Omron CX-Programmer project NewProject (CX-Programmer 9.61)

# PLC NODE_4: CS1H-H CPU67
I/O table (CPU CS1H-CPU67H): rack 0 slot 0 CS1W-ETN21(ETN21Mode); rack 0 slot 1 CS1W-PRM21; rack 0 slot 2 CS1W-PRM21; rack 0 slot 3 CS1W-PRM21; rack 0 slot 4 CS1W-PRM21

## Global symbols (name address type ; comment)
AUTOPAADRAG_P8001 D20042 UINT
AUTOPAADRAG_P8002 D20142 UINT
AUTOPAADRAG_P8003 D20242 UINT
AUTOPAADRAG_V8014 D20092 UINT
AUTOPAADRAG_V8024 D20192 UINT
AUTOPAADRAG_V8034 D20292 UINT
1052.02 BOOL  ; V8223_2_AUTO
1151.00 BOOL  ; V0941_MANUELL
1151.12 BOOL  ; V0941_MAN.COM.BIT
1151.15 BOOL  ; V0941_LUKKET
1206.00 BOOL  ; C101_IND_VST80_K2
1206.01 BOOL  ; C102_IND_VST80_K2
1206.02 BOOL  ; C103_IND_VST80_K2
1206.03 BOOL  ; C104_IND_VST80_K2
1206.04 BOOL  ; C105
1206.05 BOOL  ; C106
1206.06 BOOL  ; C107
1206.07 BOOL  ; C108
1301.15 BOOL  ; C85_CONTAINER
1321.06 BOOL  ; VST80_K3_UPROG_7
1321.07 BOOL  ; VST80_K3_UPROG_8
1350.00 BOOL  ; VST 80_K2_AUTOVASK_VALGT
1350.01 BOOL  ; VST 80_K2_AUTOVASK_NR 1 STARTER
1350.02 BOOL  ; VST 80_K2_AUTOVASK_NR 2 STARTER
1350.03 BOOL  ; VST 80_K2_AUTOVASK_NR 3 STARTER
1350.04 BOOL  ; VST 80_K2_AUTOVASK_NR 4 STARTER
1350.05 BOOL  ; VST 80_K2_AUTOVASK_NR 5 STARTER
1350.10 BOOL  ; AUTOVASK STARTER
1350.11 BOOL  ; VST 80_K2_STARTIMPULS
1350.12 BOOL  ; AUTOVASK START RESETTES
1360.00 BOOL  ; AUTOVASK ER VALGT
1360.01 BOOL  ; VST 80_K3_AUTOVASK_NR 1 STARTER
1360.02 BOOL  ; VST 80_K3_AUTOVASK_NR 2 STARTER
1360.03 BOOL  ; VST 80_K3_AUTOVASK_NR 3 STARTER
1360.04 BOOL  ; VST 80_K3_AUTOVASK_NR 4  STARTER
1360.05 BOOL  ; VST 80_K3_AUTOVASK_NR 5 STARTER
1360.10 BOOL  ; VST 80_K3_AUTOVASK START. BIT SETTES FRA GRAFIKK
1360.11 BOOL  ; VST 80_K3_STARTIMPULS
1360.12 BOOL  ; Autovask Start Resettes
1402.13 BOOL  ; LL_T82_2_LUTTANK_2
1402.14 BOOL  ; HL_T82_2 Luttank 2
2100.05 BOOL  ; P2701.01 Toemming av T27.01
2100.06 BOOL  ; P2701.02 CIP Retur
2100.09 BOOL  ; P2701.01 Fylling av T27.01
2204.13 BOOL  ; V0416_UT
2204.15 BOOL  ; V0417_UT
2211.00 BOOL  ; V0416_OE_UT
2211.01 BOOL  ; V0416_N_UT
2211.02 BOOL  ; V0517_UT
2211.03 BOOL  ; V0701.19_UT
2211.08 BOOL  ; V8223_2_UT
2211.09 BOOL  ; V8224_2_UT
2212.00 BOOL  ; V0701.02_UT
2212.01 BOOL  ; V0701.03_UT
2212.02 BOOL  ; V0701.04_UT
2212.03 BOOL  ; V0701.05_UT
2212.04 BOOL  ; V0701.06_UT
2212.05 BOOL  ; V0701.07_UT
2212.06 BOOL  ; V0701.08_UT
2212.07 BOOL  ; V0701.10_UT
2212.08 BOOL  ; V0701.11_UT
2212.09 BOOL  ; V0701.12_UT
2212.10 BOOL  ; V0701.15_UT
2212.11 BOOL  ; V0701.24_UT
2212.12 BOOL  ; V0130_UT
2212.13 BOOL  ; V0131_UT
2212.14 BOOL  ; V0132_UT
2212.15 BOOL  ; V0133_UT
2213.00 BOOL  ; V0134_UT
2213.01 BOOL  ; V0135_UT
2213.02 BOOL  ; V0136_UT
2213.03 BOOL  ; V0137_UT
2213.04 BOOL  ; V0138_UT
2213.05 BOOL  ; V0231_UT
2213.06 BOOL  ; V0232_UT
2213.07 BOOL  ; V0233_UT
2213.08 BOOL  ; V0234_UT
2213.09 BOOL  ; V0235_UT
2213.10 BOOL  ; V0236_UT
2213.11 BOOL  ; V0237_UT
2213.12 BOOL  ; V0238_UT
2213.13 BOOL  ; V0701.13_UT
2213.14 BOOL  ; V0701.09_UT
2213.15 BOOL  ; V0701.14_UT
2214.14 BOOL  ; V0516_UT
2217.14 BOOL  ; V8120_Hjelp
2226.05 BOOL  ; V0645_UT
2226.07 BOOL  ; Isvannsventil L1
2226.08 BOOL  ; Isvannsventil L2
2240.14 BOOL  ; Vannv. gr.matpumpe
2242.00 BOOL  ; V2370_UT
2242.01 BOOL  ; V2371_UT
2242.02 BOOL  ; V2372_UT
2242.03 BOOL  ; V2373_UT
2242.04 BOOL  ; V2374_UT
2242.05 BOOL  ; V2375_UT
2242.06 BOOL  ; V2376_UT
2242.07 BOOL  ; V2409_UT
2243.00 BOOL  ; V0645_UT_N5
2244.00 BOOL  ; V0316_UT
2244.01 BOOL  ; V0316_OE_UT
2244.02 BOOL  ; V0316_N_UT
2244.03 BOOL  ; V0317_UT
2244.04 BOOL  ; V0318_UT
2244.05 BOOL  ; V0132_OE_UT
2244.06 BOOL  ; V0132_N_UT
2244.07 BOOL  ; V0136_OE_UT
2244.08 BOOL  ; V0136_N_UT
2244.09 BOOL  ; V0232_OE_UT
2244.10 BOOL  ; V0232_N_UT
2244.11 BOOL  ; V0236_OE_UT
2244.12 BOOL  ; V0236_N_UT
2244.13 BOOL  ; V0701.02_OE_UT
2244.14 BOOL  ; V0701.02_N_UT
2244.15 BOOL  ; V8016_UT
2245.00 BOOL  ; V0701.16_UT
2245.01 BOOL  ; V0701.17_UT
2245.02 BOOL  ; V0701.18_UT
2245.03 BOOL  ; V0702.01_UT
2245.04 BOOL  ; V0702.02_UT
2245.05 BOOL  ; V0702.03_UT
2245.06 BOOL  ; V0702.04_UT
2245.07 BOOL  ; V0702.06_UT
2245.08 BOOL  ; V0702.07_UT
2245.09 BOOL  ; V0702.08_UT
2245.10 BOOL  ; V0702.09_UT
2245.11 BOOL  ; V0427_UT
2245.12 BOOL  ; V0437_UT
2245.13 BOOL  ; V0527_UT
2245.14 BOOL  ; V0537_UT
2245.15 BOOL  ; V0702.10_UT
2246.00 BOOL  ; V2702.01_UT
2246.01 BOOL  ; V2702.02_UT
2246.02 BOOL  ; V4021_UT
2246.03 BOOL  ; V2702.04_UT
2246.04 BOOL  ; V2702.05_UT
2246.05 BOOL  ; V2702.06_UT
2246.06 BOOL  ; V2702.07_UT
2246.07 BOOL  ; V2702.08_UT
2246.08 BOOL  ; V2702.60_UT
2246.09 BOOL  ; V2702.61_UT
2246.10 BOOL  ; V4019_UT
2246.11 BOOL  ; V2702.04_UT
2246.12 BOOL  ; V2702.04_OE_UT
2246.13 BOOL  ; V2702.04_N_UT
2246.14 BOOL  ; V2702.09_UT
2246.15 BOOL  ; V4022_UT
2247.00 BOOL  ; V2703.01_UT
2247.01 BOOL  ; V2703.02_UT
2247.02 BOOL  ; V2703.03_UT
2247.03 BOOL  ; V2703.04_UT
2247.04 BOOL  ; V2703.05_UT
2247.05 BOOL  ; V2703.06_UT
2247.06 BOOL  ; V2703.07_UT
2247.07 BOOL  ; V2703.08_UT
2247.08 BOOL  ; V2703.09_UT
2247.09 BOOL  ; V2703.60_UT
2247.10 BOOL  ; V2703.61_UT
2247.11 BOOL  ; V2713_UT
2247.12 BOOL  ; V2703.10_UT
2247.13 BOOL  ; V2703.11
2247.14 BOOL  ; V2710_OE_UT
2247.15 BOOL  ; V2710_N_UT
2252.13 BOOL  ; V0702.12_UT
2252.14 BOOL  ; V0702.13_UT
2253.07 BOOL  ; KOMM_AVL_KULEV:
2253.15 BOOL  ; KOMM_AVL_SKRAASETEV.
2256.00 BOOL  ; V0702.11_UT
2256.01 BOOL  ; V0509_UT
2256.02 BOOL  ; V0702.12_UT
2256.03 BOOL  ; V0702.13_UT
2256.04 BOOL  ; V2606_UT
2256.05 BOOL  ; V2607_UT
2256.06 BOOL  ; V2608_UT
2256.07 BOOL  ; V2609_UT
2256.08 BOOL  ; V2605_UT
2256.09 BOOL  ; V2703.12_UT
2256.10 BOOL  ; V2606_UT
2256.11 BOOL  ; V2607_UT
2256.12 BOOL  ; V2608_UT
2256.13 BOOL  ; V2609_UT
2256.14 BOOL  ; V4401_UT
2256.15 BOOL  ; V4402_UT
2257.02 BOOL  ; V0509_INN
2258.00 BOOL  ; V2702.03_UT
2258.01 BOOL  ; V2702.03_OE_UT
2258.02 BOOL  ; V2702.03_N_UT
2258.03 BOOL  ; V2702.02_N
2258.04 BOOL  ; V2702.02_OE
2258.05 BOOL  ; V2703.02_N
2258.06 BOOL  ; V2703.02_OE
2258.07 BOOL  ; V2701.01_UT
2258.08 BOOL  ; V2701.02_UT
2258.09 BOOL  ; V2701.03_UT
2258.10 BOOL  ; V2701.04_UT
2258.11 BOOL  ; V2701.05_UT
2258.12 BOOL  ; V2701.06_UT
2258.13 BOOL  ; V2701.07_UT
2258.14 BOOL  ; V2701.08_UT
2258.15 BOOL  ; V2701.09_UT
2259.00 BOOL  ; V2701.10_UT
2259.01 BOOL  ; V2701.11_UT
2259.02 BOOL  ; V2701.12_UT
2259.03 BOOL  ; V2701.60_UT
2259.04 BOOL  ; V2701.61_UT
2259.05 BOOL  ; V2701.80_UT
2259.06 BOOL  ; V2701.81_UT
2259.07 BOOL  ; V2701.02_UT_OEvre loeft
2259.08 BOOL  ; V2701.02_UT_Nedre loeft
2259.09 BOOL  ; V4506_UT
2259.10 BOOL  ; V4507_UT
2259.11 BOOL  ; V4508_UT
2292.00 BOOL  ; PLS_6_V1004.70_UT
2292.01 BOOL  ; PLS_6_V1004.71_UT
2292.02 BOOL  ; PLS_6_V1004.72_UT
2292.03 BOOL  ; PLS_6_V1004.73_UT
2292.04 BOOL  ; PLS_6_V1004.74_UT
2292.05 BOOL  ; PLS_6_V1004.75_UT
2292.06 BOOL  ; PLS_6_V1004.76_UT
2403.05 BOOL  ; STOPPE LUFTBLAASING K1
2403.06 BOOL  ; STOPP LUFTBLAASING KURS 2
2403.07 BOOL  ; Stopp P8011 Kurs 1
2403.08 BOOL  ; Stopp P8011 Kurs 2
2403.09 BOOL  ; Stopp P8012 Kurs 1
2403.10 BOOL  ; Stopp P8012 Kurs 2
2403.11 BOOL  ; Stopp P8030 Kurs 1
2403.12 BOOL  ; Stopp P8030 Kurs 2
2403.13 BOOL  ; Stopp P8031 Kurs 1
2403.14 BOOL  ; Stopp P8031 Kurs 2
2403.15 BOOL  ; KURS 1 LINJE 2.1 og 2.2
2404.05 BOOL  ; P2703.01_UT
2404.06 BOOL  ; P2703.02_UT
2404.08 BOOL  ; RV T2702_UT
2404.09 BOOL  ; RV_T2703_UT
2405.00 BOOL  ; KURS 2 LINJE 2.1 og 2.2
2501.11 BOOL  ; T82_2_HL
2504.13 BOOL  ; V0416_INN
2504.15 BOOL  ; V0417_INN
2511.00 BOOL  ; V0416_OE_INN
2511.01 BOOL  ; V0416_N_INN
2511.02 BOOL  ; V0517_INN
2511.03 BOOL  ; V0701.19_INN
2512.00 BOOL  ; V0701.02_INN
2512.01 BOOL  ; V0701.03_INN
2512.02 BOOL  ; V0701.04_INN
2512.03 BOOL  ; V0701.05_INN
2512.04 BOOL  ; V0701.06_INN
2512.05 BOOL  ; V0701.07_INN
2512.06 BOOL  ; V0701.08_INN
2512.07 BOOL  ; V0701.10_INN
2512.08 BOOL  ; V0701.11_INN
2512.09 BOOL  ; V0701.12_INN
2512.10 BOOL  ; V0701.15_INN
2512.11 BOOL  ; V0701.24_INN
2512.12 BOOL  ; V0130_INN
2512.13 BOOL  ; V0131_INN
2512.14 BOOL  ; V0132_INN
2512.15 BOOL  ; V0133_INN
2513.00 BOOL  ; V0134_INN
2513.01 BOOL  ; V0135_INN
2513.02 BOOL  ; V0136_INN
2513.03 BOOL  ; V0137_INN
2513.04 BOOL  ; V0138_INN
2513.05 BOOL  ; V0231_INN
2513.06 BOOL  ; V0232_INN
2513.07 BOOL  ; V0233_INN
2513.08 BOOL  ; V0234_INN
2513.09 BOOL  ; V0235_INN
2513.10 BOOL  ; V0236_INN
2513.11 BOOL  ; V0237_INN
2513.12 BOOL  ; V0238_INN
2513.13 BOOL  ; V0701.13_INN
2513.14 BOOL  ; V0701.09_INN
2513.15 BOOL  ; V0701.14_INN
2514.14 BOOL  ; V0516_INN
2525.02 BOOL  ; V0429_INN
2525.03 BOOL  ; V0439_INN
2525.04 BOOL  ; V0529_INN
2525.05 BOOL  ; V0539_INN
2526.05 BOOL  ; V0645_INN
2526.07 BOOL  ; Isvannsventil L1
2526.08 BOOL  ; Isvannsventil L2
2542.00 BOOL  ; V2370_AKTIVERT
2542.01 BOOL  ; V2371_AKTIVERT
2542.02 BOOL  ; V2372_AKTIVERT_INN
2542.03 BOOL  ; V2373_AKTIVERT
2542.04 BOOL  ; B2374_NEDRE
2542.05 BOOL  ; V2375_AKTIVERT
2542.06 BOOL  ; V2376_AKTIVERT
2543.00 BOOL  ; N5_V0645_INN
2544.00 BOOL  ; V0316_INN
2544.01 BOOL  ; V0316_OE_INN
2544.02 BOOL  ; V0316_N_INN
2544.03 BOOL  ; V0317_INN
2544.04 BOOL  ; V0318_INN
2544.05 BOOL  ; V0132_OE_INN
2544.06 BOOL  ; V0132_N_INN
2544.07 BOOL  ; V0136_OE_INN
2544.08 BOOL  ; V0136_N_INN
2544.09 BOOL  ; V0232_OE_INN
2544.10 BOOL  ; V0232_N_INN
2544.11 BOOL  ; V0236_OE_INN
2544.12 BOOL  ; V0236_N_INN
2544.13 BOOL  ; V0701.02_OE_INN
2544.14 BOOL  ; V0701.02_N_INN
2544.15 BOOL  ; V8016_INN
2545.00 BOOL  ; V0701.16_INN
2545.01 BOOL  ; V0701.17_INN
2545.02 BOOL  ; V0701.18_INN
2545.03 BOOL  ; V0702.01_INN
2545.04 BOOL  ; V0702.02_INN
2545.05 BOOL  ; V0702.03_INN
2545.06 BOOL  ; V0702.04_INN
2545.07 BOOL  ; V0702.06_INN
2545.08 BOOL  ; V0702.07_INN
2545.09 BOOL  ; V0702.08_INN
2545.10 BOOL  ; V0702.09_INN
2545.11 BOOL  ; V0427_INN
2545.12 BOOL  ; V0437_INN
2545.13 BOOL  ; V0527_INN
2545.14 BOOL  ; V0537_INN
2545.15 BOOL  ; V0702.10_INN
2546.00 BOOL  ; V2702.01_INN
2546.01 BOOL  ; V2702.02_INN
2546.02 BOOL  ; V4021_INN
2546.03 BOOL  ; V2702.04_INN
2546.04 BOOL  ; V2702.05_INN
2546.05 BOOL  ; V2702.06_INN
2546.06 BOOL  ; V2702.07_INN
2546.07 BOOL  ; V2702.08_INN
2546.08 BOOL  ; V2702.60_INN
2546.09 BOOL  ; V2702.61_INN
2546.10 BOOL  ; V4019_INN
2546.11 BOOL  ; V2702.04_INN
2546.14 BOOL  ; V2702.09_INN
2546.15 BOOL  ; V4022_INN
2547.00 BOOL  ; V2703.01_INN
2547.01 BOOL  ; V2703.02_INN
2547.02 BOOL  ; V2703.03_INN
2547.03 BOOL  ; V2703.04_INN
2547.04 BOOL  ; V2703.05_INN
2547.05 BOOL  ; V2703.06_INN
2547.06 BOOL  ; V2703.07_INN
2547.07 BOOL  ; V2703.08_INN
2547.08 BOOL  ; V2703.09_INN
2547.09 BOOL  ; V2703.60_INN
2547.10 BOOL  ; V2703.61_INN
2547.11 BOOL  ; V2713_INN
2547.12 BOOL  ; V2703.10_INN
2547.13 BOOL  ; V2703.11_INN
2556.00 BOOL  ; V0702.11_INN
2556.01 BOOL  ; V0509_INN
2556.02 BOOL  ; V0702.12_INN
2556.03 BOOL  ; V0702.13_INN
2556.04 BOOL  ; V2606_INN
2556.05 BOOL  ; V2607_INN
2556.06 BOOL  ; V2608_INN
2556.07 BOOL  ; V2609_INN
2556.08 BOOL  ; V2605_INN
2556.09 BOOL  ; V2703.12_INN
2556.10 BOOL  ; V2606_INN
2556.11 BOOL  ; V2607_INN
2556.12 BOOL  ; V2608_INN
2556.13 BOOL  ; V2609_INN
2556.14 BOOL  ; V4401_INN
2556.15 BOOL  ; V4402_INN
2558.00 BOOL  ; V2702.03_INN
2558.07 BOOL  ; V2701.01_INN
2558.08 BOOL  ; V2701.02_INN
2558.09 BOOL  ; V2701.03_INN
2558.10 BOOL  ; V2701.04_INN
2558.11 BOOL  ; V2701.05_INN
2558.12 BOOL  ; V2701.06_INN
2558.13 BOOL  ; V2701.07_INN
2558.14 BOOL  ; V2701.08_INN
2558.15 BOOL  ; V2701.09_INN
2559.00 BOOL  ; V2701.10_INN
2559.01 BOOL  ; V2701.11_INN
2559.02 BOOL  ; V2701.12_INN
2559.03 BOOL  ; V2701.60_INN
2559.04 BOOL  ; V2701.61_INN
2559.05 BOOL  ; V2701.80_INN
2559.06 BOOL  ; V2701.81_INN
2559.09 BOOL  ; V4506_INN
2559.10 BOOL  ; V4507_INN
2559.11 BOOL  ; V4508_INN
2592.00 BOOL  ; PLS_6_V1004.70_AKTIVERT
2592.01 BOOL  ; PLS_6_V1004.71_AKTIVERT
2592.02 BOOL  ; PLS_6_V1004.72_AKTIVERT
2592.03 BOOL  ; PLS_6_V1004.73_AKTIVERT
2592.04 BOOL  ; PLS_6_V1004.74_AKTIVERT
2592.05 BOOL  ; PLS_6_V1004.75_AKTIVERT
2592.06 BOOL  ; PLS_6_V1004.76_AKTIVERT
2605.00 BOOL  ; B2370_HJEMME
2605.01 BOOL  ; V2370_HJEMME
2605.02 BOOL  ; V2371_HJEMME
2605.03 BOOL  ; V2372_HJEMME
2605.04 BOOL  ; V2373_HJEMME
2605.05 BOOL  ; B2374_OEVRE
2605.06 BOOL  ; V2375_HJEMME
2605.07 BOOL  ; V2376_HJEMME
2605.08 BOOL  ; START GRISEFOR MOT BIL
2605.09 BOOL  ; STOPP GRISEFOR MOT BIL
2605.10 BOOL  ; NOEDSTOPP GRISEFOR MOT BIL
2605.11 BOOL  ; STOPPSIGNAL FRA FLOWMAALER GRISEFOR MOT BIL
2605.12 BOOL  ; Lampe grisefor start_stopp
2605.13 BOOL  ; Startsignal til Q4401
2607.04 BOOL  ; FEIL MAGNETROERVERK T20.37
2607.05 BOOL  ; DRIFT MAGNETROERVERK T20.37
2607.06 BOOL  ; DRIFT MAGNETROERVERK T20.36
2607.11 BOOL  ; FEIL MAGNETROERVERK T20.36
2703.03 BOOL  ; H2370
2704.06 BOOL  ; P2703.01_INN
2704.07 BOOL  ; P2703.02_INN
2704.08 BOOL  ; RV_T2702_INN
2704.09 BOOL  ; RV_T2703_INN
2704.10 BOOL  ; Drift Grundfoss-pumper
2704.11 BOOL  ; Feil paa Grundfoss-pumper
2705.05 BOOL  ; PLS 4-P1940 INN
2712.05 BOOL  ; PLS_6_H1004.70_AKTIVERT
2713.05 BOOL  ; PLS_6_B1004.70_AKTIVERT
2713.06 BOOL  ; PLS_6_B1004.71_AKTIVERT
2800.04 BOOL  ; TIL PLS 5
2817.10 BOOL  ; PLS 5-P1940 INN
2817.11 BOOL  ; PLS 5-P1940 UT
2817.12 BOOL  ; PLS 4-P2040 INN
2817.13 BOOL  ; PLS 5-P2040 UT
2817.14 BOOL  ; PLS 5-P2039 INN
2817.15 BOOL  ; PLS 5-P2039 UT
2820.15 BOOL  ; V0939_UT_TIL_PLS5
2825.00 BOOL  ; N5_V0408_OEVRE
2846.06 BOOL  ; Slange Grisefor til PLS 5
2860.00 BOOL  ; Drift_Vibrator_21.10.02
2860.01 BOOL  ; Stopp_Vibrator_21.10.02
2860.02 BOOL  ; Drift_Knuser_21.02
2860.03 BOOL  ; Stopp_Knuser_21.02
2860.04 BOOL  ; Start_stopp_Vibrator_21.10.02
2860.05 BOOL  ; Start_stopp_Knuser_21.02
2860.06 BOOL  ; Start_stopp_Utmater_21.04
2861.00 BOOL  ; Drift Vifte 21.01.01
2861.01 BOOL  ; Stopp Vifte 21.01.01
2861.02 BOOL  ; Drift Vibrator 21.01.02
2861.03 BOOL  ; Stopp Vibrator 21.01.02
2861.04 BOOL  ; Drift Vifte 21.10.01
2861.05 BOOL  ; Stopp Vifte 21.10.01
2861.06 BOOL  ; Start_stopp_Vifte_21.01.01
2861.07 BOOL  ; Start_stopp_Vibrator_21.01.02
2861.08 BOOL  ; Start_stopp_Vifte_21.10.01
2901.15 BOOL  ; N5_V0408_OEVRE
2902.02 BOOL  ; FRA_NODE_5
2902.05 BOOL  ; N5-Lavt hovedlufttrykk
2903.15 BOOL  ; PLS 4-P1940 UT
2904.04 BOOL  ; 4-RV C49
2905.13 BOOL  ; Klapr_C56
2905.15 BOOL  ; Klapr_C92
2919.06 BOOL  ; 5-Bypass Mikronisator
2919.07 BOOL  ; 5-2919.07
2919.08 BOOL  ; 5-2919.08
2919.09 BOOL  ; 5-2919.09
2919.10 BOOL  ; 5-2919.10
2923.13 BOOL  ; N5_V2006_UT
2935.06 BOOL  ; V4302_UT_N5
2935.13 BOOL  ; V4302 Forsinkelse
2937.01 BOOL  ; 5-P2040_UT
2940.00 BOOL  ; N5_T20.36 Tapping
2940.01 BOOL  ; N5_T20.37 Tapping
2941 CHANNEL  ; N5_NIVAA_T2036
2944 CHANNEL  ; N5_NIVAA_T20.37
2946.00 BOOL  ; Retn.1 fra N5
2946.01 BOOL  ; Retn.2 fra N5
2946.02 BOOL  ; Isv.alarm fra N5
2955.07 BOOL  ; OPEN_DREN
2955.08 BOOL  ; OPEN_DYREFOR
2956.07 BOOL  ; OPEN_DREN_26
2956.08 BOOL  ; OPEN_DYREFOR_26
2959.00 BOOL  ; N5_V0408_OEVRE
302.13 BOOL  ; C106_VALG
302.14 BOOL  ; C107_VALG
4813.13 BOOL  ; TRYKKOMSLAG DP3 SPERRET
5117 CHANNEL  ; PT L1-1
5118 CHANNEL  ; PT L1-2
5119 CHANNEL  ; PT L2-1
5161.03 BOOL  ; .
5172 CHANNEL  ; TT T07.01
5173 CHANNEL  ; PT T07.01
5174 CHANNEL  ; TT T07.02
5175 CHANNEL  ; PT T07.02
5432.02 BOOL  ; Lampe drift grisefortoemming
5588 CHANNEL  ; TEMP_T82_2
5589 CHANNEL  ; Temp Kommunalt avloep
5590 CHANNEL  ; PH Kommunalt avloep
5591 CHANNEL  ; Flow Kommunalt avloep
5592 CHANNEL  ; BRIX Kommunalt avloep
5593 CHANNEL  ; PT T82_2
5594 CHANNEL  ; B8203_2
5595 CHANNEL  ; B8016
5596 CHANNEL  ; B8026
5597 CHANNEL  ; B8036
5601.02 BOOL  ; ¨
5667.03 BOOL  ; ¨
5730.00 BOOL  ; 360802
5761.02 BOOL  ; ,
5824.04 BOOL  ; '
587.00 BOOL  ; PGM587_DRIFT
587.01 BOOL  ; PGM587_0-STATUS
587.02 BOOL  ; PGM587_1-STATUS
587.03 BOOL  ; PGM587_2-STATUS
587.04 BOOL  ; PGM587_FEIL
587.05 BOOL  ; PGM587_FEILTID
587.06 BOOL  ; PGM587_INDKON
587.07 BOOL  ; PGM587_START
587.09 BOOL  ; PGM587_STOPP
587.10 BOOL  ; PGM587_STARTIMP.
587.11 BOOL  ; PGM587_ONIMPULS
587.14 BOOL  ; PGM587_OFFIMPULS
587.15 BOOL  ; PGM587_IND.INNE
588.00 BOOL  ; PGM 588 DRIFT
588.01 BOOL  ; 0-Status PGM 588
588.02 BOOL  ; PGM 588 1-Status
588.03 BOOL  ; PGM 588 2-Status
588.04 BOOL  ; PGM 588 FEIL
588.05 BOOL  ; PGM 588 Feiltid
588.06 BOOL  ; PGM 588_IndKon
588.07 BOOL  ; PGM 588 START
588.09 BOOL  ; PGM 588_STOPP
588.11 BOOL  ; PGM 588_Onimpuls
588.14 BOOL  ; PGM 588_Offimpuls
588.15 BOOL  ; PGM 588 Individkontroll
589.00 BOOL  ; PGM 589_DRIFT
589.01 BOOL  ; PGM 589 0-Status
589.02 BOOL  ; PGM 589 1-Status
589.03 BOOL  ; PGM 589_2-Status
589.04 BOOL  ; PGM 589_FEIL
589.05 BOOL  ; PGM589_FEILTID
589.06 BOOL  ; PGM 589_INDKON
589.07 BOOL  ; PGM 589_START
589.09 BOOL  ; PGM 589_STOPP
589.11 BOOL  ; PGM 589_ONIMPULS
589.14 BOOL  ; PGM 589_Offimpuls
589.15 BOOL  ; PGM 589_INDIVIDKONTROLL
590.00 BOOL  ; PGM 590 DRIFT
590.01 BOOL  ; 0-Status PGM 590
590.02 BOOL  ; 1-Status PGM 590
590.03 BOOL  ; PGM 590 2-Status
590.04 BOOL  ; PGM 590 FEIL
590.05 BOOL  ; PGM 590 Feiltid
590.06 BOOL  ; PGM 590 IndKon
590.07 BOOL  ; PGM 590 Start
590.09 BOOL  ; PGM 590_STOPP
590.11 BOOL  ; PGM 590 ONIMPULS
590.14 BOOL  ; PGM 590 Offimpuls
590.15 BOOL  ; PGM 590 Individkontroll
591.00 BOOL  ; PGM 591 DRIFT
591.01 BOOL  ; PGM 591 0-Status
591.02 BOOL  ; PGM 591 1-Status
591.03 BOOL  ; PGM 591_2-Status
591.04 BOOL  ; PGM 591 FEIL
591.05 BOOL  ; PGM 591 Feiltid
591.06 BOOL  ; PGM 591_IndKon
591.07 BOOL  ; PGM 591_START
591.09 BOOL  ; PGM 591_STOPP
591.11 BOOL  ; PGM 591_Onimpuls
591.14 BOOL  ; PGM 591_Offimpuls
591.15 BOOL  ; PGM 591_Individkontroll
592.00 BOOL  ; PGM 592_DRIFT
592.01 BOOL  ; PGM 592 0-Status
592.02 BOOL  ; PGM 592 1-Status
592.03 BOOL  ; PGM 592 2-Status
592.04 BOOL  ; PGM 592 FEIL
592.05 BOOL  ; PGM 592 Feiltid
592.06 BOOL  ; PGM 592_IndKon
592.07 BOOL  ; PGM 592 Start
592.09 BOOL  ; PGM 592_FEILTID
592.11 BOOL  ; PGM 592_Onimpuls
592.14 BOOL  ; PGM 592_Offimpuls
592.15 BOOL  ; PGM 592_Individkontroll
593.00 BOOL  ; PGM 593 DRIFT
593.01 BOOL  ; PGM 593 0-Status
593.02 BOOL  ; PGM 593_1-Status
593.03 BOOL  ; PGM 593_2-Status
593.05 BOOL  ; PGM 593_Feiltid
593.06 BOOL  ; PGM 593 IndKon
593.07 BOOL  ; PGM 593_START
593.09 BOOL  ; PGM 593_STOPP
593.11 BOOL  ; PGM 593 Onimpuls
593.14 BOOL  ; PGM 593_Offimpuls
593.15 BOOL  ; PGM 593 Individkontroll
600.02 BOOL  ; Drenering C33
608.04 BOOL  ; UHT-Anlegg mot Dypvannsutslipp
609.00 BOOL  ; RV2703Y
609.01 BOOL  ; RV2703I
609.02 BOOL  ; T2703_Vasket
609.03 BOOL  ; T2703_ManStartet
609.04 BOOL  ; T27.02_Sperr
609.05 BOOL  ; T27.03_Sperr
609.06 BOOL  ; P270301_ManStartet
609.07 BOOL  ; P270302_ManStartet
609.08 BOOL  ; P270201_ManStartet
609.09 BOOL  ; T2702_Vasket
609.10 BOOL  ; P070201_ManStartet
609.11 BOOL  ; P270201_I
609.12 BOOL  ; P270201_Y
609.13 BOOL  ; RV2702Y
609.14 BOOL  ; RV2702I
609.15 BOOL  ; Manuell Ansep CIP
610.00 BOOL  ; RV2702_ManStartet
610.01 BOOL  ; T0702_Vasket
610.02 BOOL  ; RV2703_ManStartet
610.03 BOOL  ; Start PGM 591.00
610.04 BOOL  ; Start PGM 589.00
610.05 BOOL  ; Start PGM 588.00
610.06 BOOL  ; Start PGM 590.00
610.07 BOOL  ; RV2703Y
610.09 BOOL  ; Dren til Silo 3
610.10 BOOL  ; Dren til Silo 4
610.11 BOOL  ; Dren til Silo 5
610.12 BOOL  ; Hj1_V0516
610.13 BOOL  ; Hj1_V0416
610.14 BOOL  ; Hj1_V0316
610.15 BOOL  ; Hj1_B0701.11
611.00 BOOL  ; Bil 1_Silo 3
611.01 BOOL  ; Bil 1_Silo 4
611.02 BOOL  ; Bil 1_Silo 5
611.03 BOOL  ; Henger 1_Silo 3
611.04 BOOL  ; Henger 1_Silo 4
611.05 BOOL  ; Henger 1_Silo 5
611.06 BOOL  ; Bil 2_Silo 3
611.07 BOOL  ; Bil 2_Silo 4
611.08 BOOL  ; Bil 2_Silo 5
611.09 BOOL  ; Henger 2_Silo 3
611.10 BOOL  ; Henger 2_Silo 4
611.11 BOOL  ; Henger 2_Silo 5
611.12 BOOL  ; Hj1_Dren til Silo 3
611.13 BOOL  ; Hj1_Drenering fra T0701 til Silo 4
611.14 BOOL  ; Hj1_Drenering fra T0701 til Silo 5
611.15 BOOL  ; Start PGM 592.00
612.03 BOOL  ; Vannsp_T27.02_Start
612.04 BOOL  ; Vannsp_T27.02_Drift
612.05 BOOL  ; Vannsp_T27.02_Feil
612.06 BOOL  ; Vannsp_T27.03_Start
612.07 BOOL  ; Vannsp_T27.03_Drift
612.08 BOOL  ; Vannsp_T27.03_Feil
612.09 BOOL  ; Vannsp_T27.40_Start
612.10 BOOL  ; Vannsp_T27.40_Drift
612.11 BOOL  ; Vannsp_T27.40_Feil
612.12 BOOL  ; Vannsp_T27.41_Start
612.13 BOOL  ; Vannsp_T27.41_Drift
612.14 BOOL  ; Vannsp_T27.41_Feil
612.15 BOOL  ; Manuell testbryter
613.00 BOOL  ; PGM 588 Hj1
613.01 BOOL  ; Start PGM 593.00
613.02 BOOL  ; PGM 592 Hj1
613.03 BOOL  ; Toerrkj. P4501
613.04 BOOL  ; Overtrykk, stopp griseforpumpe
613.05 BOOL  ; Hj1_Overtrykk gr_pumpe
613.06 BOOL  ; Makstid VST80 KURS 1
613.07 BOOL  ; Makstid for VST80 KURS 2
613.08 BOOL  ; Makstid utloept VST80 KURS 3
613.09 BOOL  ; Hj1_Autovask_80K3
613.10 BOOL  ; Hj2_Autovask_80K3
613.11 BOOL  ; Hj3_Autovask_80K3
613.12 BOOL  ; Hj4_Autovask_80_K3
613.13 BOOL  ; Hj5_Autovask_80K3
613.15 BOOL  ; PGM501_KOMMANDO_KOE
614.09 BOOL  ; Hj1_Autovask_80K2
614.10 BOOL  ; Hj2_Autovask_80K2
614.12 BOOL  ; Hj4_Autovask_80K2
614.13 BOOL  ; Hj5_Autovask_80K2
614.14 BOOL  ; Sperr innlesning til koeregister
614.15 BOOL  ; PGM 502 KOMMANDO_KOE
615.00 BOOL  ; Hj._0-Status_C101,C102
615.01 BOOL  ; Hj.1-Status_C101
615.02 BOOL  ; Hj.1-Status_C102
615.03 BOOL  ; PGM587_VALG
615.04 BOOL  ; Hj1_PGM587
615.05 BOOL  ; Hj2_PGM587
615.06 BOOL  ; Hj3_PGM587
615.07 BOOL  ; Hj4_PGM587
615.08 BOOL  ; Hj5_PGM587
615.09 BOOL  ; Hj6_PGM587
615.10 BOOL  ; Hj7_PGM587_Steg 1
615.11 BOOL  ; Hj8_PGM587_Steg 2
615.12 BOOL  ; Hj9_PGM587_Steg 3
615.13 BOOL  ; Hj10_PGM587_Steg 4
615.14 BOOL  ; Dren T27.01 til T20.33-35
615.15 BOOL  ; Slangefeil Trakt UHT
616.00 BOOL  ; PGM502_IND_C106_VALG
616.01 BOOL  ; PGM502_IND_C107_VALG
616.02 BOOL  ; PGM 589_VALG
616.03 BOOL  ; Hj1_PGM589
616.04 BOOL  ; Hj2_PGM589
616.05 BOOL  ; Hj3_PGM589
616.06 BOOL  ; Hj4_PGM589
616.07 BOOL  ; Hj5_PGM589
616.10 BOOL  ; PGM502_IND_C33_VALG
616.11 BOOL  ; C33_Drenert
616.12 BOOL  ; C33_Vasket
616.13 BOOL  ; C33_Hj1
616.14 BOOL  ; C33_Hj2
616.15 BOOL  ; Hj1_C14_V0582
617.00 BOOL  ; Hj.1_1-Status_C103
617.01 BOOL  ; Hj.2_1-Status_C104
617.02 BOOL  ; Hj.3_1-Status_C104
617.03 BOOL  ; Hj.4_1-Status_C104
617.04 BOOL  ; T07.01_Sperr
617.05 BOOL  ; T07.02_Sperr
617.06 BOOL  ; PGM 591_VALG
617.07 BOOL  ; Hj1_PGM 591
617.08 BOOL  ; Hj2_PGM 591
617.09 BOOL  ; Hj3_PGM 591
617.10 BOOL  ; Hj4_PGM 591
617.11 BOOL  ; Hj5_PGM 591
617.12 BOOL  ; PGM 592_VALG
617.13 BOOL  ; PGM 593_VALG
617.14 BOOL  ; PGM588_VALG
618.00 BOOL  ; Stopp fra FT Q2703
618.01 BOOL  ; Noedstopp fra Panel Deponi
618.02 BOOL  ; Stoppknapp Panel Deponi
618.03 BOOL  ; Startknapp Panel Deponi
618.04 BOOL  ; Lampe Drift Panel Deponi
618.05 BOOL  ; Startsignal til FT Q2703
618.06 BOOL  ; Hj.4_1-Status_C104
618.07 BOOL  ; Hj.5_1-Status C104
618.12 BOOL  ; Hj1_T0701_Sperr
618.13 BOOL  ; Hj2_T0701_Sperr
618.14 BOOL  ; Hj1_T0702_Sperr
618.15 BOOL  ; Hj2_T0702_Sperr
619.00 BOOL  ; Ny morgendrenering aktivert
619.01 BOOL  ; Dren L1.1 Til Silo 3
619.02 BOOL  ; Dren L1.1 Til Silo 4
619.03 BOOL  ; Dren L1.1 Til Silo 5
619.04 BOOL  ; Dren L1.2 Til Silo 3
619.05 BOOL  ; Dren L1.2 Til Silo 4
619.06 BOOL  ; Dren L1.2 Til Silo 5
619.07 BOOL  ; Dren L2.1 Til Silo 3
619.08 BOOL  ; Dren L2.1 Til Silo 4
619.09 BOOL  ; Dren L2.1 Til Silo 5
619.10 BOOL  ; Dren L2.2 Til Silo 3
619.11 BOOL  ; Dren L2.2 Til Silo 4
619.12 BOOL  ; Dren L2.2 Til Silo 5
619.13 BOOL  ; Kveldsdrenering Startet
619.14 BOOL  ; Nivaa i T0701 over SP
620.00 BOOL  ; Kveldsdrenering L1.1 Startet
620.01 BOOL  ; Kveldsdrenering L1.2 Startet
620.02 BOOL  ; Kveldsdrenering L2.1 Startet
620.03 BOOL  ; Kveldsdrenering L2.2 Startet
620.04 BOOL  ; Morgendrenering utfoert L1.1
620.05 BOOL  ; Morgendrenering utfoert L1.2
620.06 BOOL  ; Morgendrenering utfoert L2.1
620.07 BOOL  ; Morgendrenering utfoert L2.2
620.08 BOOL  ; Morgendrenering Turbiditet L1.1 over SP
620.09 BOOL  ; Morgendrenering Turbiditet L1.2 over SP
620.10 BOOL  ; Morgendrenering Turbiditet L2.1 over SP
620.11 BOOL  ; Morgendrenering Turbiditet L2.2 over SP
620.12 BOOL  ; Kveldsdrenering utfoert L1.1
620.13 BOOL  ; Kveldsdrenering utfoert L1.2
620.14 BOOL  ; Kveldsdrenering utfoert L2.1
620.15 BOOL  ; Kveldsdrenering utfoert L2.2
621.00 BOOL  ; Hj1_PGM 590
621.01 BOOL  ; Hj2_PGM 590
621.02 BOOL  ; Hj3_PGM 590
621.03 BOOL  ; Hj4_PGM 590
621.04 BOOL  ; Hj5_PGM 590
621.05 BOOL  ; Hj2_PGM592
621.06 BOOL  ; Hj3_PGM 592
621.07 BOOL  ; Hj4_PGM 592
621.08 BOOL  ; Hj5_PGM 592
621.09 BOOL  ; Hj6_PGM 592
621.10 BOOL  ; Hj1_PGM 593
621.11 BOOL  ; Hj2_PGM 593
621.12 BOOL  ; Hj3_PGM 593
621.13 BOOL  ; Hj4_PGM 593
621.14 BOOL  ; Hj4_PGM 593
622.00 BOOL  ; Hj1_PGM 588
622.01 BOOL  ; Hj3_PGM 588
622.02 BOOL  ; Hj4_PGM 588
622.03 BOOL  ; Hj5_PGM 588
622.04 BOOL  ; Hj1_L1.1_Kveldsdrenering
622.05 BOOL  ; Hj1_L1.2_Kveldsdrenering
622.06 BOOL  ; Hj1_L2.1_Kveldsdrenering
622.07 BOOL  ; Hj1_L2.2_Kveldsdrenering
622.08 BOOL  ; Hj1_Toem_T07.01
622.09 BOOL  ; Toem T07.02
622.10 BOOL  ; Test_3
622.11 BOOL  ; Flow OK VST80 K1
622.13 BOOL  ; UHT Trakt Prioritet
622.14 BOOL  ; 80K2_timingOK
622.15 BOOL  ; 80K3_timingOK
623.00 BOOL  ; Avloepstank 1 Mottak Overloep
623.01 BOOL  ; Avloepstank 1 Mottak HL
623.02 BOOL  ; Avloepstank 1 Mottak LL
623.03 BOOL  ; Avloepstank 1 Mottak Drift
623.04 BOOL  ; Avloepstank 1 Mottak Pumpe 1
623.05 BOOL  ; Avloepstank 1 Mottak Pumpe 2
623.06 BOOL  ; Avloepstank 1 Mottak Overloepsvarsel
623.07 BOOL  ; Avloepstank 2 Mottak Kjeller Overloep
623.08 BOOL  ; Avloepstank 2 Mottak Kjeller HL
623.09 BOOL  ; Avloepstank 2 Mottak Kjeller LL
623.10 BOOL  ; Avloepstank 2 Mottak Kjeller Drift
623.11 BOOL  ; Avloepstank 2 Mottak Kjeller Pumpe 3
623.12 BOOL  ; Avloepstank 2 Mottak Kjeller Overloepsvarsel
623.13 BOOL  ; Feil paa en frekvensomformer kommunalt avloep
623.14 BOOL  ; Reset makstemp dypvannsutslipp
623.15 BOOL  ; Reset doegntid
624.00 BOOL  ; Ny Kveldsdrenering aktivert
624.01 BOOL  ; Dren utfoert, toem T07.01
624.02 BOOL  ; T07.01 toemt, vanndren mot Silo
624.03 BOOL  ; Nye drenering C33 aktivert
624.04 BOOL  ; Kveldsdrenering Turbiditet L1.1 under SP
624.05 BOOL  ; Kveldsdrenering Turbiditet L1.2 under SP
624.06 BOOL  ; Kveldsdrenering Turbiditet L2.1 under SP
624.07 BOOL  ; Kveldsdrenering Turbiditet L2.2 under SP
624.08 BOOL  ; Morgendrenering L1.1 Startet
624.09 BOOL  ; Morgendrenering L1.2 Startet
624.10 BOOL  ; Morgendrenering L2.1 Startet
624.11 BOOL  ; Morgendrenering L2.2 Startet
624.12 BOOL  ; Hj1_Kveldsdrenering L1.1
624.13 BOOL  ; Hj1_Kveldsdrenering L1.2
624.14 BOOL  ; Hj1_Kveldsdrenering L2.1
624.15 BOOL  ; Hj1_Kveldsdrenering L2.2
625.01 BOOL  ; C106_Hj1
625.02 BOOL  ; Nye drenstart L1.1
625.03 BOOL  ; Nye drenstart L1.2
625.04 BOOL  ; Nye drenstart L2.1
625.05 BOOL  ; Nye drenstart L2.2
625.06 BOOL  ; Kveldsdren mot Silo 3
625.07 BOOL  ; Kveldsdren mot Silo 4
625.08 BOOL  ; Kveldsdren mot Silo 5
625.09 BOOL  ; Autodren Raamelkslinjer og Batteri
625.12 BOOL  ; Hurtigvask VST80_K2
625.13 BOOL  ; Hurtigvask VST80_K3
625.14 BOOL  ; Autovask_K3_Av_Paa
625.15 BOOL  ; Autovask K2_Av_Paa
626.00 BOOL  ; Makstid morgendrenering L1.1
626.01 BOOL  ; Makstid Moprgendrenering L1.2
626.02 BOOL  ; Makstid Morgendrenering L2.1
626.03 BOOL  ; Makstid Morgendrenering L2.2
626.04 BOOL  ; PGM501_IND_C102_VALG
626.05 BOOL  ; PGM501_IND_C101_VALG
626.06 BOOL  ; PGM501_IND_C06_VALG
626.07 BOOL  ; PGM501_IND_C103_VALG
626.08 BOOL  ; PGM501_IND_C104_VALG
626.09 BOOL  ; PGM501_IND_C105_VALG
626.10 BOOL  ; PGM501_IND_C108_VALG
626.11 BOOL  ; PGM501_IND_C53_VALG
626.12 BOOL  ; PGM501_IND_C54_VALG
626.13 BOOL  ; PGM501_IND_C77_VALG
626.14 BOOL  ; PGM501_IND_C78_VALG
626.15 BOOL  ; PGM501_IND_C79_VALG
627.00 BOOL  ; PGM502_IND_C12_VALG
627.01 BOOL  ; PGM502_IND_C13_VALG
627.02 BOOL  ; PGM502_IND_C14_VALG
627.03 BOOL  ; PGM502_IND_C30_VALG
627.04 BOOL  ; PGM502_IND_C09_VALG
627.05 BOOL  ; PGM502_IND_C10_VALG
627.06 BOOL  ; PGM502_IND_C15_VALG
628.00 BOOL  ; VST80_K1_Trinn 2 Turbiditet
628.01 BOOL  ; VST80_K2_Trinn 2 Turbiditet
628.02 BOOL  ; VST80_K3_Trinn 2_Turbiditet
628.03 BOOL  ; Nivaa i T07.02 OK
628.04 BOOL  ; T27.03 Vasket
628.05 BOOL  ; C104 Vasket
628.06 BOOL  ; Deponi-roer drenert
628.07 BOOL  ; T07.02 Vasket
628.08 BOOL  ; RV T07.01 Vasket
628.09 BOOL  ; T07.01 Vasket
628.10 BOOL  ; T27.02 Vasket
628.11 BOOL  ; PGM592_Hj1
628.12 BOOL  ; Isvann Hoey Temp Retning 1
628.13 BOOL  ; Isvann Hoey Temp Retning 2
628.14 BOOL  ; Hj5_V8221
628.15 BOOL  ; Hj6_V8221
629.00 BOOL  ; Autovask_K2_Hj1
629.01 BOOL  ; Autovask K3 Hj1
629.02 BOOL  ; C102 Vasket
629.03 BOOL  ; Autovask K2 Hj1
629.04 BOOL  ; V4202_Hj1
629.05 BOOL  ; Turbiditet i forskyll K1
629.06 BOOL  ; Turbiditet i forskyll K2
629.07 BOOL  ; Turbiditet i forskyll K3
629.08 BOOL  ; Hj.4_VST80K3
629.09 BOOL  ; Hj.5_VST80K3
630.00 BOOL  ; Dren batteri L1.1
630.01 BOOL  ; Dren batteri L1.2
630.02 BOOL  ; Dren batteri L2.1
630.03 BOOL  ; Dren batteri L2.2
630.04 BOOL  ; Start drenering av batteri
630.05 BOOL  ; Batteri L1.1 i drenering
630.06 BOOL  ; Batteri L1.2 i drenering
630.07 BOOL  ; Batteri L2.1 i drenering
630.08 BOOL  ; Batteri L2.2 i drenering
630.13 BOOL  ; T82_2_Hj1
630.14 BOOL  ; T82_2_Hj2
630.15 BOOL  ; T82_2_SPERRING
631.00 BOOL  ; Kveldsdrenering_Start_L2.1
631.01 BOOL  ; L2_1_Startknapp
631.02 BOOL  ; L2.1 Drenering Startet
631.03 BOOL  ; L2.1 Drenering Utfoert
631.04 BOOL  ; L2.1 Vann i Linje
631.05 BOOL  ; L2.1 Melk i Linje
631.06 BOOL  ; Kveldsdrenering_Start_L2.2
631.07 BOOL  ; L2.2 Startknapp
631.08 BOOL  ; L2.2 Drenering Startet
631.09 BOOL  ; L2.2 Drenering Utfoert
631.10 BOOL  ; L2.2 Vann i Linje
631.11 BOOL  ; L2.2 Melk i Linje
631.13 BOOL  ; Start Drenering C33
631.14 BOOL  ; Drenering C33 Startet
631.15 BOOL  ; Drenering C33 Utfoert
632.00 BOOL  ; Kveldsdrenering_Start_L1.1
632.01 BOOL  ; L1_1_Startknapp
632.02 BOOL  ; L1.1 Drenering Startet
632.03 BOOL  ; L1.1 Drenering Utfoert
632.04 BOOL  ; L1.1 Vann i Linje
632.05 BOOL  ; L1.1 Melk i Linje
632.06 BOOL  ; Kveldsdrenering_Start_L1.2
632.07 BOOL  ; L1_2_Startknapp
632.08 BOOL  ; L1_2_Startet
632.09 BOOL  ; L1.2 Drenering Utfoert
632.10 BOOL  ; L1.2 Vann i Linje
632.11 BOOL  ; L1.2 Melk i Linje
632.12 BOOL  ; Vann i Linje C33
632.13 BOOL  ; Melk i Linje C33
633.00 BOOL  ; L1.1_Dren_Hj1
633.01 BOOL  ; L1.1_Dren_Hj2
633.02 BOOL  ; L1.2_Dren_Hj1
633.03 BOOL  ; L1.2_Dren_Hj2
633.04 BOOL  ; L2.1_Dren_Hj1
633.05 BOOL  ; L2.1_Dren_Hj2
633.06 BOOL  ; L2.2 Dren_Hj1
633.07 BOOL  ; L2.2_Dren_Hj2
633.08 BOOL  ; Dren L1.1 under batteri
633.09 BOOL  ; Dren L1.2 under batteri
633.10 BOOL  ; Dren L2.1 under batteri
633.11 BOOL  ; Dren L2.2 under batteri
633.12 BOOL  ; Dren L1.1 batteri utfoert
633.13 BOOL  ; Dren L1.2 batteri utfoert
633.14 BOOL  ; Dren L2.1 batteri utfoert
633.15 BOOL  ; Dren L2.2 batteri utfoert
634.00 BOOL  ; C33_Dren_1-Status_Hj1
634.01 BOOL  ; C33_Dren_1-Status_Hj2
634.02 BOOL  ; C33_Dren_2-Status_Hj3
634.03 BOOL  ; C33_Dren_2-Status_Hj4
634.04 BOOL  ; Drenkontroll_L1.1
634.05 BOOL  ; Drenkontroll_L1.2
634.06 BOOL  ; Drenkontroll_L2.1
634.07 BOOL  ; Drenkontroll_L2.2
634.08 BOOL  ; Drenkontroll_C33
634.09 BOOL  ; C33 i drift
634.10 BOOL  ; V0701.20_UT
634.11 BOOL  ; V0701.20_INN
634.12 BOOL  ; Forsinkelse LL T07.01
634.13 BOOL  ; Manuell kjoering V2161 Damp Pasteur 21
634.14 BOOL  ; Floetepumpe P26.01_Inn
634.15 BOOL  ; Floetepumpe P26.01 UT
635.00 BOOL  ; C33_Dren_1-Status Hj4
635.01 BOOL  ; C33_Dren_1-Status Hj5
635.02 BOOL  ; C33_Dren_1-Status Hj6
635.03 BOOL  ; Dren_Batteri
635.04 BOOL  ; Dren_Linjer
635.05 BOOL  ; T0701_Drift_Drenering
635.06 BOOL  ; Turbiditet_Over_SP L1.1
635.07 BOOL  ; Turbiditet_Over_SP_L1.2
635.08 BOOL  ; Turbiditet_Over_SP_L2.1
635.09 BOOL  ; Turbiditet_Over_SP_L2.2
635.10 BOOL  ; Ok aa drenere batteriet
635.11 BOOL  ; Ok aa drenere Linjene
635.12 BOOL  ; Makstid drenering L1.1
635.13 BOOL  ; Makstid for drenering L1.2
635.14 BOOL  ; Makstid for drenering L2.1
635.15 BOOL  ; Makstid for drenering L2.2
636.00 BOOL  ; Rele' drift til P2040
636.01 BOOL  ; P2040 Drift
636.02 BOOL  ; P1940 Drift
636.03 BOOL  ; Griseforpumpe P1940 Start
636.04 BOOL  ; Griseforpumpe manuell hast.
636.05 BOOL  ; P2040 Manuell hast.
636.06 BOOL  ; Floetepumpe P2039 Manuell hast.
636.07 BOOL  ; P2039_UT
636.08 BOOL  ; Start slange grisefor
636.09 BOOL  ; Slangedrift Skummesal
636.10 BOOL  ; Start slange grisefor 1-status
636.11 BOOL  ; Start slange grisefor 2-status
636.12 BOOL  ; V9026_UT
636.13 BOOL  ; V9026_INN
638.00 BOOL  ; Toerrkjoerings-sperre for P0101 ved toemming av tankbil L1.1
638.01 BOOL  ; Toerrkjoerings-sperre for P0111 ved toemming av tankbil L1.2
638.02 BOOL  ; Toerrkjoerings-sperre for P0201 ved toemming av tankbil L2.1
638.03 BOOL  ; Toerrkjoerings-sperre for P0211 ved toemming av tankbil L2.2
639.09 BOOL  ; Hj1_RV_T27.02
639.12 BOOL  ; St_Kjoeling_T27.02
639.13 BOOL  ; St_Kjoeling_T27.03
639.14 BOOL  ; Ok aa starte kjoeling T27.02
639.15 BOOL  ; Ok aa starte kjoeling T27.03
641.02 BOOL  ; 1-Status L1.1
641.03 BOOL  ; 2 Status L1.1
641.04 BOOL  ; Fe_L1.1_Silo
641.05 BOOL  ; Feiltid_L1.1_Silo
641.07 BOOL  ; StL1.1_Silo
641.11 BOOL  ; Fe_Drenbatteri_L1.1
641.12 BOOL  ; DrenStBatteri_L1.1
641.13 BOOL  ; DrenBatteri_L1.1
641.14 BOOL  ; S1Batteri_L1.1
641.15 BOOL  ; S2Batteri_L1.1
642.02 BOOL  ; 1-Status L1.1
642.03 BOOL  ; 2-Status L1.2
642.04 BOOL  ; Fe_L1.2_Silo
642.05 BOOL  ; Feiltid_L1.2_Silo
642.07 BOOL  ; StL1.2_Silo
642.11 BOOL  ; Fe_Drenbatteri_L1.2
642.12 BOOL  ; DrenStBatteri_L1.2
642.13 BOOL  ; DrenBatteri_L1.2
642.14 BOOL  ; S1Batteri_L1.2
642.15 BOOL  ; S2Batteri_L1.2
643.02 BOOL  ; 1-Status L2.1
643.03 BOOL  ; 2-Status L2.1
643.04 BOOL  ; Fe_L2.1_Silo
643.05 BOOL  ; Feiltid_L2.1
643.07 BOOL  ; StL2.1_Silo
643.11 BOOL  ; Fe_Drenbatteri_L2.1
643.12 BOOL  ; DrenStBatteri_L2.1
643.13 BOOL  ; DrenBatteri_L2.1
643.14 BOOL  ; S1Batteri_L2.1
643.15 BOOL  ; S2Batteri_L2.1
644.02 BOOL  ; 1-Status L2.2
644.03 BOOL  ; 2-Status L2.2
644.04 BOOL  ; Fe_L2.2_Silo
644.05 BOOL  ; Feiltid_L2.2
644.07 BOOL  ; StL2.2_Silo
644.11 BOOL  ; Fe_Drenbatteri_L2.2
644.12 BOOL  ; DrenStBatteri_L2.2
644.13 BOOL  ; DrenBatteri_L2.2
644.14 BOOL  ; S1Batteri_L2.2
644.15 BOOL  ; S2Batteri_L2.2
645.00 BOOL  ; Turbiditet over setpunkt
645.01 BOOL  ; Start dren L1.2
645.02 BOOL  ; Start dren L2.1
645.03 BOOL  ; Start dren L2.2
645.08 BOOL  ; Hj1_0-Status Batteri L1.1
645.09 BOOL  ; Hj1_0-Status Batteri L1.2
645.10 BOOL  ; Hj1_0-Status Batteri L2.1
645.11 BOOL  ; Hj1_0-Status Batteri L2.2
645.12 BOOL  ; Start autodren L1.1
645.13 BOOL  ; Start autodren L1.2
645.14 BOOL  ; Start autodren L2.1
645.15 BOOL  ; Start autodren L2.2
646.00 BOOL  ; Hj1_0-Status L1.1
646.01 BOOL  ; Hj2_0-Status L1.1
646.02 BOOL  ; Hj3_0-Status L1.1
646.03 BOOL  ; Hj1_1-Status L1.1
646.04 BOOL  ; Hj2_1-Status L1.1
646.05 BOOL  ; Hj3_1-Status L1.1
646.06 BOOL  ; Hj4_1-Status L1.1
646.07 BOOL  ; Hj1_2-Status L1.1
646.08 BOOL  ; Hj1_0-Status L1.2
646.09 BOOL  ; Hj2_0-Status L1.2
646.10 BOOL  ; Hj3_0-Satus L1.2
646.11 BOOL  ; Hj1_1-Status L1.2
646.12 BOOL  ; Hj2_1-Status L1.2
646.13 BOOL  ; Hj3_1-Status L1.2
646.14 BOOL  ; Hj4_1-Status L1.2
646.15 BOOL  ; Hj1_2-Status L1.2
647.00 BOOL  ; Hj1_0-Status L2.1
647.01 BOOL  ; Hj2_0-Status L2.1
647.02 BOOL  ; Hj3_0-Status L2.1
647.03 BOOL  ; Hj1_1-Status L2.1
647.04 BOOL  ; Hj2_1-Status L2.1
647.05 BOOL  ; Hj3_1-Status L2.1
647.06 BOOL  ; Hj4_1-Status L2.1
647.07 BOOL  ; Hj1_2-Status L2.1
647.08 BOOL  ; Hj1_0-Status L2.2
647.09 BOOL  ; Hj2_0-Status L2.2
647.10 BOOL  ; Hj3_0-Status L2.2
647.11 BOOL  ; Hj1_1-Status L2.2
647.12 BOOL  ; Hj2_1-Status L2.2
647.13 BOOL  ; Hj3_1-Status L2.2
647.14 BOOL  ; Hj4_1-Status L2.2
647.15 BOOL  ; Hj1_2-Status L2.2
650.04 BOOL  ; Hj.Ind.Inne_2_80K2
650.05 BOOL  ; C101_VALG_VST80K2
650.06 BOOL  ; C102_VALG_VST80K2
650.07 BOOL  ; C103_VALG_VST80_K2
650.08 BOOL  ; C104_VALG_VST80_K2
650.09 BOOL  ; C105_VALG_VST80_K2
650.10 BOOL  ; C108_VALG_VST80_K2
650.15 BOOL  ; Lavt damptrykk
651.02 BOOL  ; 1 status
651.03 BOOL  ; 2 status
651.04 BOOL  ; feil
651.07 BOOL  ; Roed blink
659.00 BOOL  ; Dr_Autodren
659.01 BOOL  ; S0_Autodren
659.02 BOOL  ; S1_Autodren
659.03 BOOL  ; S2_Autodren
659.04 BOOL  ; Fe_Autodren
659.07 BOOL  ; St_Autodren
659.08 BOOL  ; Feiltid_Batteridrenering L1.1
659.09 BOOL  ; Feiltid_Batteridrenering_L1.2
659.10 BOOL  ; Feiltid_Batteridrenering_L2.1
659.11 BOOL  ; Feiltid_Batteridrenering_L2.2
659.12 BOOL  ; Hj1_T0701_Drift
659.14 BOOL  ; Hj2_Autodren
659.15 BOOL  ; Hj1_Autodren
660.00 BOOL  ; St_Overpumping_Til_T27.02
660.02 BOOL  ; S1_Overpumping_Til_T27.02
660.03 BOOL  ; S2_Overpumping_Til_T27.02
660.04 BOOL  ; Fe_Overpumping_Til_T27.02
660.05 BOOL  ; Dr_Overpumping_T27.02
660.06 BOOL  ; St_Overpumping_Til_T27.03
660.08 BOOL  ; S1_Overpumping_Til_T27.03
660.09 BOOL  ; S2_Overpumping_Til_T27.03
660.10 BOOL  ; Fe_Overpumping_Til_T27.03
660.11 BOOL  ; Dr_Overpumping_Til_T27.03
660.12 BOOL  ; Dren_Toem luftutskiller L1.1
660.13 BOOL  ; Dren_Toem luftutskiller L1.2
660.14 BOOL  ; Dren_Luftutskiller L2.1
660.15 BOOL  ; Dren_Luftutskiller L2.2
661.02 BOOL  ; S1_Kjoeling_T27.02
661.03 BOOL  ; S2_Kjoeling_T27.02
661.04 BOOL  ; Fe_Kjoeling_T27.02
661.05 BOOL  ; Dr_Kjoeling_T27.02
661.08 BOOL  ; S1_Kjoeling_T27.03
661.09 BOOL  ; S2_Kjoeling_T27.03
661.10 BOOL  ; Fe_Kjoeling_T27.03
661.11 BOOL  ; Dr_Kjoeling_T27.03
661.12 BOOL  ; T27.02 i koe
661.13 BOOL  ; T27.02 koe-start
661.14 BOOL  ; T27.03 i koe
661.15 BOOL  ; T27.03 i koe-start
662.00 BOOL  ; V2702.08_UT
662.01 BOOL  ; V2703.13_UT
662.02 BOOL  ; V2703.14_UT
662.03 BOOL  ; V2702.08_INN
662.04 BOOL  ; V2703.13_INN
662.05 BOOL  ; V2703.14_INN
662.06 BOOL  ; Turbiditet over min. VST80 Luttank
677.01 BOOL  ; AV_PAA_PIGGING
724.00 BOOL  ; T20.36 Tapping
724.01 BOOL  ; T20.37 Tapping
724.02 BOOL  ; Nivaa T20.36 mellom 40 og 50 000 liter
724.03 BOOL  ; Nivaa T20.36 mellom 30 og 40 000 liter
724.04 BOOL  ; Nivaa T20.36 mellom 25 og 30 000 liter
724.05 BOOL  ; Nivaa T20.36 mellom 20 og 25 000 liter
724.06 BOOL  ; Nivaa T20.36 mellom 6 og 20 000 liter
724.07 BOOL  ; Nivaa T20.37 mellom 40 og 50 000 liter
724.08 BOOL  ; Nivaa T20.37 mellom 30 og 40 000 liter
724.09 BOOL  ; Nivaa T20.37 mellom 25 og 30 000 liter
724.10 BOOL  ; Nivaa T20.37 mellom 20 og 25 000 liter
724.11 BOOL  ; Nivaa T20.37 mellom 6 og 20 000 liter
724.12 BOOL  ; Nivaa T20.36 under 6 000 liter stopp roerverk
724.13 BOOL  ; Nivaa T20.37 under 6 000 stopp roerverk
800.04 BOOL  ; Man Bactofors P2301
800.07 BOOL  ; C106 HJ1
800.08 BOOL  ; C107 HJ1
800.09 BOOL  ; C106 HJ 2
800.10 BOOL  ; C106 HJ3
800.12 BOOL  ; C107 HJ3
800.13 BOOL  ; C107 HJ4
800.14 BOOL  ; C106 HJ4
800.15 BOOL  ; C107 HJ5
801.00 BOOL  ; P0501_HJ5
801.07 BOOL  ; MANUELL KNAPP
802.00 BOOL  ; Manuell toemming silo
802.01 BOOL  ; Fra silo 3
802.02 BOOL  ; Fra silo 4
802.03 BOOL  ; Fra silo 5
802.04 BOOL  ; Til silo 3
802.05 BOOL  ; Til silo 4
802.06 BOOL  ; Til silo 5
803.00 BOOL  ; Ferdig sterilisert
803.01 BOOL  ; Ferdig sterilisert
803.02 BOOL  ; Ferdig sterilisert
803.03 BOOL  ; Trykkomslag_Pasteur 21
803.04 BOOL  ; Trykkomslag_Pasteur 22
803.05 BOOL  ; Trykkomslag_Pasteur 23
810.00 BOOL  ; Forsinkelse utloept Past.21 DP1
810.01 BOOL  ; Start forsinkelse Past.21 DP1
810.02 BOOL  ; Forsinkelse utloept Past.21 DP2
810.03 BOOL  ; Start forsinkelse Past.21 DP2
810.04 BOOL  ; Forsinkelse utloept Past.22 DP1
810.05 BOOL  ; Start forsinkelse Past.22 DP1
810.06 BOOL  ; Forsinkelse utloept Past.22 DP2
810.07 BOOL  ; Start forsinkelse Past.22 DP2
810.08 BOOL  ; Forsinkelse utloept Past.22 DP3
810.09 BOOL  ; Start forsinkelse Past. 22 DP3
810.10 BOOL  ; Reset tellere omslag pasteurer
820.00 BOOL  ; PLS_6_V1004.70_DEAKTIVERT
820.01 BOOL  ; PLS_6_V1004.71_DEAKTIVERT
820.02 BOOL  ; PLS_6_V1004.72_DEAKTIVERT
820.03 BOOL  ; PLS_6_V1004.73_DEAKTIVERT
820.04 BOOL  ; PLS_6_V1004.74_DEAKTIVERT
820.05 BOOL  ; PLS_6_V1004.75_DEAKTIVERT
820.06 BOOL  ; PLS_6_V1004.76_DEAKTIVERT
821.00 BOOL  ; P0701.01_UT
821.01 BOOL  ; V2371_DEAKTIVERT
821.02 BOOL  ; V2372_DEAKTIVERT
821.03 BOOL  ; V2373_DEAKTIVERT
821.04 BOOL  ; V2374_DEAKTIVERT
821.05 BOOL  ; V2375_DEAKTIVERT
821.06 BOOL  ; V2376_DEAKTIVERT
821.07 BOOL  ; B2370_INN
821.09 BOOL  ; V4302_UT_N5
821.10 BOOL  ; V4202 Forsinkelse
822.00 BOOL  ; Lampe omslag past.21
822.01 BOOL  ; Lampe omslag past.22
822.02 BOOL  ; Lampe omslag past.23
822.03 BOOL  ; Vannventil P2304
823.00 BOOL  ; Start P0701.01
823.01 BOOL  ; Drift P0701.01
823.02 BOOL  ; Oppheve sperring kurs 1
823.03 BOOL  ; Oppheve sperring kurs 2
823.05 BOOL  ; HL T07.01
823.06 BOOL  ; Start P0702.01
823.07 BOOL  ; LL T07.01
823.08 BOOL  ; HL T07.02
823.09 BOOL  ; LL T07.02
823.10 BOOL  ; Driftsignal fra P0702.01
823.11 BOOL  ; Motorvern P0702.01
904.03 BOOL  ; 0
905.09 BOOL  ; Man Bactofors
905.10 BOOL  ; Man Bactofors P2304
905.11 BOOL  ; Man Bactofors P2101
905.12 BOOL  ; Man Bactofors P2104
905.13 BOOL  ; Man Bactofors P2201
905.14 BOOL  ; Man Bactofors P2204
909.03 BOOL  ; Proeveuttak kommunalt avloep
925.10 BOOL  ; Toemming grisefortank til bil
925.15 BOOL  ; Telling ferdig fra flowmaaler Q4401
941.04 BOOL  ; HJ1_V8223_2_AUT
953.14 BOOL  ; ¨
955.13 BOOL  ; ¨
962.07 BOOL  ; Startknapp slange skummesal
962.08 BOOL  ; Start slange Grisefor Skummesal
962.09 BOOL  ; Drift Slange Grisefor Skummesal
964.11 BOOL  ; Manuell reset
964.12 BOOL  ; Manuell reset
964.13 BOOL  ; Test flowmaaler VST80 K3
965.00 BOOL  ; Man.sirk. Isv.tank
966.00 BOOL  ; FLOW KURS 1 OK
966.01 BOOL  ; FLOW K2 OK
966.02 BOOL  ; FLOW K3 OK
967.00 BOOL  ; VST80_K2_AUTOVASK
967.01 BOOL  ; Hjelpebit  VST80_K2_AUTOVASK
967.02 BOOL  ; Hjelpebit VST80_K2_AUTOVASK
967.05 BOOL  ; Hjelpebit VST 80_K3_AUTOVASK
967.06 BOOL  ; Hjelpebit VST 80_K3_AUTOVASK
967.07 BOOL  ; Hjelpebit VST 80_K3_AUTOVASK
969.00 BOOL  ; HJ_1_V8224_2
972.00 BOOL  ; OPEN_V4210
972.01 BOOL  ; OPEN_V4211
972.02 BOOL  ; OPEN_V4218
972.04 BOOL  ; OPEN_V4219
C0135 BOOL  ; Makstid for drenering C33 til T07.01
C0136 BOOL  ; Makstid Drenering C33
C0137 BOOL  ; Makstid Toem T07.01
C0138 BOOL  ; Makstid Vanndren mot Silo
C0139 BOOL  ; Holdetid foer Turbiditet er ute
C0231 BOOL  ; Drenstid L1.1
C0232 BOOL  ; Drenstid L1.2
C0233 BOOL  ; Drenstid L2.1
C0234 BOOL  ; Drenstid L2.2
C0235 BOOL  ; Forsink reset drenering av batteri
C0236 BOOL  ; Drenstid L1.1
C0237 BOOL  ; Drenstid Batteri L1.1
C0238 BOOL  ; Drenstid L1.2
C0239 BOOL  ; Drenstid Batteri L1.2
C0240 BOOL  ; Drenstid L2.1
C0241 BOOL  ; Drenstid Batteri L2.1
C0242 BOOL  ; Drenstid L2.2
C0243 BOOL  ; Drenstid Batteri L2.2
C0244 BOOL  ; Feiltid_Overpumping til T27.02
C0245 BOOL  ; Feiltid_Overpumping_Til_T27.03
C0246 BOOL  ; Feiltid_Kjoeling_T27.02
C0257 BOOL  ; Hindre toerrkjoering for P0101
C0258 BOOL  ; Hindre toerrkjoering for P0111
C0259 BOOL  ; Hindre toerrkjoering for P0201
C0260 BOOL  ; Hindre toerrkjoering for P0211
C0261 BOOL  ; RV T27.02 Intervall Stopp
C0262 BOOL  ; RV T27.02 Intervall Drift
C0263 BOOL  ; RV T27.03 Intervall Stopp
C0264 BOOL  ; RV T27.03 Intervall Drift
C0351 BOOL  ; Doegnreset for dypvannstemp
C0684 BOOL  ; Klapreteller C79
C0685 BOOL  ; Klapreteller
C0686 BOOL  ; PAUSETID KOMMUNAL SPYLING
C0687 BOOL  ; FORSINKELSE SKRAASETEVENTIL
C0688 BOOL  ; SPYLETID BRIXMAALER KOMMUNALT AVLOEP
C0690 BOOL  ; SEKUNDER AAPEN MOT DYPVANNSUTSLIPP TELLER NED FRA 3600
C0691 BOOL  ; TIMER AAPEN MOT DYPVANNSUTSLIPP TELLER NED FRA 3600
C0692 BOOL  ; SEKUNDER FYLLEVENTIL V0655 ER AAPEN PAA VANNSPARETANK
C0693 BOOL  ; TIMER FYLLEVENTIL V0655 ER AAPEN PAA VANNSPARETANK
C0715 BOOL  ; Makstid for vask utloept
C0716 BOOL  ; Makstid for vask utloept
C0717 BOOL  ; Makstid for vask utloept
C135 CHANNEL  ; Makstid til T07.01 sendes til Historian
C351 CHANNEL  ; Doegnteller dypvannsutslipp
D10148 CHANNEL  ; Skalering for bruk av Historian
D10154 CHANNEL  ; Skalering for bruk i Historian
D11101 CHANNEL  ; P
D11102 CHANNEL  ; I
D11103 CHANNEL  ; D
D15003 CHANNEL  ; Node 4.03
D15004 CHANNEL  ; Node 4.04
D15005 CHANNEL  ; Node 4.05
D15006 CHANNEL  ; Node 4.06
D15007 CHANNEL  ; Node 4.07
D15008 CHANNEL  ; Node 4.08
D15009 CHANNEL  ; Node 4.09
D15010 CHANNEL  ; Node 4.10
D15011 CHANNEL  ; Node 4.11
D15012 CHANNEL  ; Node 4.12
D15013 CHANNEL  ; Node 4.13
D15014 CHANNEL  ; Node 4.14
D15015 CHANNEL  ; Node 4.15
D15028 CHANNEL  ; Slavefeil Bus 4
D15029 CHANNEL  ; Diagnosefeil Bus 4
D15031 CHANNEL  ; Node 5.01
D15032 CHANNEL  ; Node 5.02
D15033 CHANNEL  ; Node 5.03
D15034 CHANNEL  ; Node 5.04
D15035 CHANNEL  ; Node 5.05
D15036 CHANNEL  ; Node 5.06
D15037 CHANNEL  ; Node 5.07
D15038 CHANNEL  ; Node 5.08
D15039 CHANNEL  ; Node 5.09
D15040 CHANNEL  ; Node 5.10
D15041 CHANNEL  ; Node 5.11
D15042 CHANNEL  ; Node 5.12
D15043 CHANNEL  ; Node 5.13
D15044 CHANNEL  ; Node 5.14
D15045 CHANNEL  ; Node 5.15
D15046 CHANNEL  ; Node 5.16
D15047 CHANNEL  ; Node 5.17
D15048 CHANNEL  ; Node 5.18
D15049 CHANNEL  ; Node 5.19
D15050 CHANNEL  ; Node 5.20
D15058 CHANNEL  ; Slavefeil Bus 5
D15059 CHANNEL  ; Diagnosefeil Bus 5
D15062 CHANNEL  ; Node 3.02
D15063 CHANNEL  ; Node 3.03
D15088 CHANNEL  ; Slavefeil Bus 3
D15089 CHANNEL  ; Diagnosefeil Bus 3
D15091 CHANNEL  ; Node 2.01
D15092 CHANNEL  ; Node 2.02
D15093 CHANNEL  ; Node 2.03
D15094 CHANNEL  ; Node 2.04
D15095 CHANNEL  ; Node 2.05
D15096 CHANNEL  ; Node 2.06
D15097 CHANNEL  ; Node 2.07
D15098 CHANNEL  ; Node 2.12
D15099 CHANNEL  ; Node 2.13
D15100 CHANNEL  ; Node 2.14
D15101 CHANNEL  ; Node 2.15
D15102 CHANNEL  ; Node 2.16
D15103 CHANNEL  ; Node 2.17
D15104 CHANNEL  ; Node 2.18
D15105 CHANNEL  ; Node 2.19
D15106 CHANNEL  ; Node 2.20
D15107 CHANNEL  ; Node 2.21
D15108 CHANNEL  ; Node 2.22
D15109 CHANNEL  ; Node 2.23
D15110 CHANNEL  ; Node 2.24
D15111 CHANNEL  ; Node 2.25
D15112 CHANNEL  ; Node 2.26
D15113 CHANNEL  ; Node 2.27
D15118 CHANNEL  ; Slavefeil Bus 2
D15119 CHANNEL  ; Diagnosefeil Bus 2
D1658 CHANNEL  ; Temp Kommunalt avloep
D1660 CHANNEL  ; PH Kommunalt avloep
D1662 CHANNEL  ; Flow Kommunalt avloep
D1664 CHANNEL  ; Brix Kommunalt avloep
D1750 CHANNEL  ; Turbiditet retur kurs 1
D17500 CHANNEL  ; Turbiditet retur kurs 1
D1752 CHANNEL  ; Turbiditet retur kurs 2
D17520 CHANNEL  ; Turbiditet retur kurs 2
D1754 CHANNEL  ; Turbiditet retur kurs 3
D1756 CHANNEL  ; Turbiditet retur kurs 3
D196 CHANNEL  ; D3174
D4032 CHANNEL  ; TEMP DYPVANNSUTSLIPP
D4034 CHANNEL  ; SKALERING
D4036 CHANNEL  ; SKALERT VERDI FOR TEMP DYPVANNSUTSLIPP
D4374 CHANNEL  ; Turbiditetsmaaler Raamelkslinje 2.2 Skalert
D4376 CHANNEL  ; Linje 2.2 Skalert verdi
D4380 CHANNEL  ; Turbiditetsmaaler Raamelkslinje 1.1
D4382 CHANNEL  ; Turbiditet Raamelkslinje 1.1
D4384 CHANNEL  ; Linje 1.1 Skalert verdi
D4386 CHANNEL  ; Turbiditetsmaaler Raamelkslinje 1.2
D4388 CHANNEL  ; Turbiditetsmaaler Raamelkslinje 1.2 Skalert
D4390 CHANNEL  ; Linje 1.2 Skalert verdi
D4392 CHANNEL  ; Turbiditetsmaaler Raamelkslinje 2.1
D4394 CHANNEL  ; Turbiditesmaaler Raamelkslinje 2.1 Skalert
D4396 CHANNEL  ; Linje 2.1 Skalert verdi
D4398 CHANNEL  ; Turbiditetsmaaler Raamelkslinje 2.2
D4400 CHANNEL  ; Turbiditetsmaaler Raamelkslinje 2.2 Skalert
D4402 CHANNEL  ; Linje 2.2 Skalert verdi
D4408 CHANNEL  ; Hastighet P0701.01
D4411 CHANNEL  ; B07.01.03
D4412 CHANNEL  ; B07.01.04
D4413 CHANNEL  ; B07.02.03
D4414 CHANNEL  ; B07.02.04
D4427 CHANNEL  ; NIVAA T07.02
D4434 CHANNEL  ; PT L1-1 B0107
D4440 CHANNEL  ; PT L1-2 B0117
D4446 CHANNEL  ; PT L2-1 B0207
D4452 CHANNEL  ; PT L2-2 B0217
D4458 CHANNEL  ; PT ISVANN L1 B0108
D4464 CHANNEL  ; PT ISVANN L2 B0208
D4466 CHANNEL  ; TRYKKDIFF L1.1
D4468 CHANNEL  ; TRYKKDIFF L1.2
D4470 CHANNEL  ; TRYKKDIFF L2.1
D4472 CHANNEL  ; TRYKKDIFF L2.2
D4474 CHANNEL  ; B07.01.04
D4500 CHANNEL  ; VST 80_K2_AUTOVASK FELLESREGISTER
D4501 CHANNEL  ; VST 80_K2_AUTOV_CNR_V1
D4502 CHANNEL  ; VST 80_K2_AUTOV_CNR_V2
D4503 CHANNEL  ; VST 80_K2_AUTOV_CNR_V3
D4504 CHANNEL  ; VST 80_K2_AUTOV_CNR_V4
D4505 CHANNEL  ; VST 80_K2_AUTOV_CNR_V5
D4600 CHANNEL  ; VST 80_K3_AUTOVASK FELLESREGISTER
D4601 CHANNEL  ; VST 80_K3_AUTOV_CNR_V1
D4602 CHANNEL  ; VST 80_K3_AUTOV_CNR_V2
D4603 CHANNEL  ; VST 80_K3_AUTOV_CNR_V3
D4604 CHANNEL  ; VST 80_K3_AUTOV_CNR_V4
D4605 CHANNEL  ; VST 80_K3_AUTOV_CNR_V5
D4700 CHANNEL  ; Temp Kommunalt avloep til Panel verksted
D4702 CHANNEL  ; pH Kommunalt avloep til Panel verksted
D4704 CHANNEL  ; Flow kommunalt avloep til Panel verksted
D4706 CHANNEL  ; Brix Kommunalt avloep til Panel Verksted
D4708 CHANNEL  ; Nivaa i Vannsparetank til Panel Verksted
D4710 CHANNEL  ; Flow Vannsparetank til Panel Verksted
D4712 CHANNEL  ; Makstemp dypvannsutslipp
D4714 CHANNEL  ; Mintemp dypvannsutslipp
D4716 CHANNEL  ; Resttid foer autoreset dypvannsutslipp
D5016 CHANNEL  ; PGM501_KOEPLASS_4
D5018 CHANNEL  ; PGM501_KOEPLASS_5
D5026 CHANNEL  ; PGM502_KOEPLASS_4
D5028 CHANNEL  ; PGM502_KOEPLASS_5
D5030 CHANNEL  ; Verdi C0302 til Historian
D5130 CHANNEL  ; 80K3_Vask_Dag
D5132 CHANNEL  ; 80K3_Vask_Mnd
D5134 CHANNEL  ; 80K3_Vask_Time
D5136 CHANNEL  ; 80K3_Vask_Min
D5138 CHANNEL  ; 80K2_Vask_Dag
D5140 CHANNEL  ; 80K2_Vask_Mnd
D5142 CHANNEL  ; 80K2_Vask_Time
D5144 CHANNEL  ; 80K2_Vask_Min
D5146 CHANNEL  ; Fellesregister for tidspunkt
D5300 CHANNEL  ; Bil 1
D5302 CHANNEL  ; Henger 1
D5304 CHANNEL  ; Bil 2
D5306 CHANNEL  ; Henger 2
D5432 CHANNEL  ; TT B0103
D5436 CHANNEL  ; TT B0104
D5502 CHANNEL  ; Status til Dreamreport
D5504 CHANNEL  ; Status til Dreamreport
D6052 CHANNEL  ; D6026
D6290 CHANNEL  ; Sperrekode for T07.01
D6291 CHANNEL  ; Kode aktivert T07.01
D6292 CHANNEL  ; Sperrekode for T07.02
D6293 CHANNEL  ; Kode aktivert T07.02
D6294 CHANNEL  ; Sperrekode for T27.02
D6295 CHANNEL  ; Kode aktivert T27.02
D6296 CHANNEL  ; Sperrekode for T27.03
D6297 CHANNEL  ; Kode aktivert T27.03
D6300 CHANNEL  ; Nivaa Avloepstank 1 Mottak
D6302 CHANNEL  ; Avloepstank 2 Mottak Kjeller Nivaa
D6304 CHANNEL  ; TT T27.02
D6308 CHANNEL  ; TT T27.02
D6310 CHANNEL  ; TT T27.03
D6312 CHANNEL  ; D6314
D6314 CHANNEL  ; TT T27.03
D6336 CHANNEL  ; P20.39 Hastighet
D6400 CHANNEL  ; Man Hast P2101 Bactofors
D6402 CHANNEL  ; Man Hast P2104 Bactofors
D6404 CHANNEL  ; Man Hast P2201 Bactofors
D6406 CHANNEL  ; Man Hast P2204 Bactofors
D6408 CHANNEL  ; Man Hast P2301 Bactofors
D6410 CHANNEL  ; Man Hast P2304 Bactofors
D6514 CHANNEL  ; B2106
D6530 CHANNEL  ; B2108
D6546 CHANNEL  ; P21_Diff_1
D6562 CHANNEL  ; P21_Diff_2
D6594 CHANNEL  ; B2330
D6614 CHANNEL  ; B2206
D6630 CHANNEL  ; B2208
D6646 CHANNEL  ; P22_Diff_1
D6662 CHANNEL  ; P22_Diff_2
D6678 CHANNEL  ; P22_Diff_3
D6694 CHANNEL  ; P22_Diff_ISv.
D6714 CHANNEL  ; B2306
D6730 CHANNEL  ; B2308
D6746 CHANNEL  ; P23_Diff_1
D6762 CHANNEL  ; P23_Diff_2
D6778 CHANNEL  ; P23_Diff_3
D6794 CHANNEL  ; P23_Diff_Isv.
D6800 CHANNEL  ; Hastighet P2040
D6806 CHANNEL  ; Hastighet P2040
D6808 CHANNEL  ; Hastighet P1940
D6900 CHANNEL  ; Hastighet P1940
D6902 CHANNEL  ; Skalert hastighet P1940
D7004 CHANNEL  ; Turbiditet VST80 Luttank
D7008 CHANNEL  ; Skalert verdi Turbiditet VST80 Luttank
D7716 CHANNEL  ; C101_TYPE_VASK
D7717 CHANNEL  ; C102_TYPE_VASK
D7718 CHANNEL  ; C103_TYPE_VASK
D7719 CHANNEL  ; C104_TYPE_VASK
D7736 CHANNEL  ; VASKESTATUS C101
D7737 CHANNEL  ; VASKESTATUS C102
D7738 CHANNEL  ; VASKESTATUS C103
D7739 CHANNEL  ; VASKESTATUS C104
D7741 CHANNEL  ; C105_TYPE_VASK
D7742 CHANNEL  ; C_TYPE_VASK
D7743 CHANNEL  ; C108_TYPE_VASK
D8080 CHANNEL  ; ID nummer fra Bil Kurs 1
D8082 CHANNEL  ; ID nummer fra Henger Kurs 1
D8084 CHANNEL  ; ID nummer fra Bil Kurs 2
D8086 CHANNEL  ; ID nummer fra Henger Kurs 2
D8090 CHANNEL  ; Bil Kurs 1
D8092 CHANNEL  ; Henger Kurs 1
D8094 CHANNEL  ; Bil 2
D8096 CHANNEL  ; Henger 2
D8250 CHANNEL  ; T82_2_SPERR_KODE_INN
D8251 CHANNEL  ; D82_2_SPERR_KODE_UT
D9012 CHANNEL  ; T82_2_ER_TEMP
D9016 CHANNEL  ; T82_2_NIVAA
D9018 CHANNEL  ; T82_2_NIVAA
D9430 CHANNEL  ; VASKESTATUS
D9432 CHANNEL  ; VASKESTATUS
T0158 BOOL  ; Feiltid Start Autodren
T0182 BOOL  ; Vent foer Turbiditet er ute
T0183 BOOL  ; Vent foer Turbiditet er ute
T0184 BOOL  ; Vent foer Turbiditet er ute
T0211 BOOL  ; Makstid for morgendrenering L1.1
T0212 BOOL  ; Makstid for morgendrenering L1.2
T0213 BOOL  ; Makstid for morgendrenering L2.1
T0214 BOOL  ; Makstid for morgendrenering L2.2
T0215 BOOL  ; Makstid for kveldsdrenering L1.1
T0216 BOOL  ; Makstid for kveldsdrenering L1.2
T0217 BOOL  ; Makstid for kveldsdrenering L2.1
T0218 BOOL  ; Makstid for kveldsdrenering L2.2
T0219 BOOL  ; Forsinkelse Turbiditet L1.1
T0220 BOOL  ; Forsinkelse Turbiditet L1.2
T0221 BOOL  ; Forsinkelse Turbiditet L2.1
T0222 BOOL  ; Forsinkelse Turbiditet L2.2
T0223 BOOL  ; Forsinkelse Turbiditet Kveldsdrenering L1.1
T0224 BOOL  ; Forsinkelse Turbiditet Kveldsdrenering L1.2
T0225 BOOL  ; Forsinkelse Turbiditet Kveldsdrenering L2.1
T0226 BOOL  ; Forsinkelse Turbiditet Kveldsdrenering L2.2
T0237 BOOL  ; V4202 Forsinkelse
T0242 BOOL  ; Hold foer stenging av V4205
T0243 BOOL  ; Hold foer stenging av V4202
T0252 BOOL  ; C33_Hj2_Forsink_Ut
T0253 BOOL  ; Makstid_Drenering_T07.01
T0254 BOOL  ; B2106
T0255 BOOL  ; B2108
T0256 BOOL  ; P21_Diff_1
T0257 BOOL  ; P21_Diff_2
T0258 BOOL  ; P21_Diff_Isv.
T0259 BOOL  ; B2206
T0260 BOOL  ; B2208
T0261 BOOL  ; P22_Diff_1
T0262 BOOL  ; P22_Diff_2
T0263 BOOL  ; P22_Diff_3
T0264 BOOL  ; P22_Diff_Isv.
T0265 BOOL  ; B2306
T0266 BOOL  ; B2308
T0267 BOOL  ; P23_Diff_1
T0268 BOOL  ; P23_Diff_2
T0269 BOOL  ; P23_Diff_3
T0270 BOOL  ; P23_Diff_Isv.
T0273 BOOL  ; Forsinkelse turbiditetskontroll
T0274 BOOL  ; Forsinkelse turbiditetskontroll
T0275 BOOL  ; Forsinkelse turbiditetskontroll
T0276 BOOL  ; Forsinkelse turbiditetskontroll
T0278 BOOL  ; Makstid drenering til T27.02/T27.03
T0279 BOOL  ; Makstid drenering L1.1
T0280 BOOL  ; Makstid drenering L1.2
T0281 BOOL  ; Makstid drenering L2.1
T0282 BOOL  ; Makstid drenering L2.2
T0283 BOOL  ; Dren L1.1 batteri makstid
T0284 BOOL  ; Dren L1.2 batteri makstid
T0285 BOOL  ; Dren L2.1 batteri makstid
T0286 BOOL  ; Dren L2.2 batteri makstid
T0287 BOOL  ; Forsinkelse LL T07.01
T0305 BOOL  ; Tid etter ventil stenger
T0306 BOOL  ; Tid etter ventil stenger
T0307 BOOL  ; Tid etter ventil stenger
T0308 BOOL  ; Tid etter ventil stenger
T0312 BOOL  ; Feiltid L1.1
T0313 BOOL  ; Feiltid Batteridrenering L1.1
T0314 BOOL  ; Feiltid L1.2
T0315 BOOL  ; Feiltid Batteridrenering L1.2
T0316 BOOL  ; Feiltid L2.1
T0317 BOOL  ; Feiltid Batteridrenering L2.1
T0318 BOOL  ; Feiltid L2.2
T0319 BOOL  ; Feiltid Batteridrenering L2.2
T0706 BOOL  ; Autovask forsinker startimpuls
T0731 BOOL  ; Maks tid aapen for V0701.10
T0732 BOOL  ; PGM587 FEILTID
T0734 BOOL  ; PGM 589 FEILTID
T0735 BOOL  ; PGM 593 FEILTID
T0736 BOOL  ; Fra T07.01 mot Silo 3, Drenstid
T0737 BOOL  ; Fra T07.01 mot Silo 4, Drenstid
T0738 BOOL  ; Fra T07.01 mot Silo 5, Drenstid
T0787 BOOL  ; PGM 588 Feiltid
T0847 BOOL  ; Drenering fra T0701 til Silo 3
T0848 BOOL  ; Drenering fra T0701 til Silo 4
T0849 BOOL  ; Drenering fra T0701 til Silo 5
T0850 BOOL  ; Spyletid paa V0701.07
T0975 BOOL  ; Dreneringstid Deponi
T0976 BOOL  ; TID OVERTRYKK GRISEFORPUMPE
T0977 BOOL  ; TID IKKE OVERTRYKK GRISEFORPUMPE
B0101_0_1000 D2004 REAL  ; 0=0GRADER   1000=100.0 GRADER
B0101_HJREG1 D6138 REAL
B0101_TT D1714 REAL  ; ZZ
B0102_0_1000 D2006 REAL  ; 0=0GRADER   1000=100.0 GRADER
B0102_HJREG1 D6140 REAL
B0102_TT D1694 REAL  ; Z
B0103_FC 2602.00 BOOL  ; Z
B0103_TT_ISVTUR D2044 WORD  ; TUR ISVANSTEMP TIL MOTTAK SKALERT
B0103_TT_ISVTUR_RAA D1724 WORD  ; TUR ISVANSTEMP TIL MOTTAK
B0104_TT_ISVRETUR D2046 WORD  ; RETUR ISVANSTEMP FRA MOTTAK SKALERT
B0104_TT_ISVRETUR_RAA D1726 WORD  ; RETUR ISVANSTEMP FRA MOTTAK
B0105_HL 2600.08 BOOL  ; Z
B0106_LL 2602.04 BOOL  ; Z
B0106_ML 2602.05 BOOL  ; Z
B0111_0_1000 D2104 REAL  ; 0=0GRADER   1000=100.0 GRADER
B0111_HJREG1 D6142 REAL
B0111_TT D1716 REAL  ; ZZ
B0112TT D1700 REAL  ; Z
B0112_0_1000 D2106 REAL  ; 0=0GRADER   1000=100.0 GRADER
B0112_HJREG1 D6144 REAL
B0113_FC 2602.01 BOOL  ; Z
B0115_HL 2600.09 BOOL  ; Z
B0116_LL 2602.06 BOOL  ; Z
B0116_ML 2602.07 BOOL  ; Z
B0201_0_1000 D2204 REAL  ; 0=0GRADER   1000=100.0 GRADER
B0201_HJREG1 D6146 REAL
B0201_TT D1718 REAL  ; ZZ
B0202_0_1000 D2206 REAL  ; 0=0GRADER   1000=100.0 GRADER
B0202_HJREG1 D6148 REAL
B0202_TT D1706 REAL  ; Z
B0203_FC 2602.02 BOOL  ; Z
B0205_HL 2600.10 BOOL  ; Z
B0206_LL 2602.08 BOOL  ; Z
B0206_ML 2602.09 BOOL  ; Z
B0211_0_1000 D2304 REAL  ; 0=0GRADER   1000=100.0 GRADER
B0211_HJREG1 D6150 REAL
B0211_TT D1720 REAL  ; ZZ
B0212_0_1000 D2306 REAL  ; 0=0GRADER   1000=100.0 GRADER
B0212_HJREG1 D6152 REAL
B0212_TT D1712 REAL  ; Z
B0213_FC 2602.03 BOOL  ; Z
B0215_HL 2600.11 BOOL  ; Z
B0216_LL 2602.10 BOOL  ; Z
B0216_ML 2602.11 BOOL  ; Z
B0301_LL 2600.13 BOOL  ; Z
B0302_TT_T03 D1730 WORD  ; INNGANGS0RD TEMP.
B0303_PT_T03 D1732 WORD  ; INNGANGSORD NIVAA
B0303_TT D6000 CHANNEL  ; Z
B0304_PT D6002 CHANNEL  ; Z
B0351_FC 2601.00 BOOL  ; Z
B0361_FC 2601.01 BOOL  ; Z
B0401_LL 2600.01 BOOL  ; Z
B0402_HL 2600.00 BOOL  ; Z
B0403_PT_T04 D1722 WORD  ; INNGANGSORD NIVAA
B0403_TT D6020 CHANNEL  ; Z
B0403_TT_INN D1748 REAL
B0404_PT D6022 CHANNEL  ; Z
B0404_PT_MAALT D6046 INT
B0501_LL 2600.03 BOOL  ; Z
B0502_TT_T05 D1740 WORD  ; INNGANGS0RD TEMP.
B0503_PT_T05 D1742 WORD  ; INNGANGSORD NIVAA
B0503_TT D6040 CHANNEL  ; Z
B0504_PT D6042 CHANNEL  ; Z
B0504_PT_MAALT D6026 INT
B0510_FC 2601.09 BOOL  ; Z
B0601_PT D6064 INT
B0603_PT_T06 D1746 CHANNEL
B0604_LL 2601.12 BOOL
B0605_FLOW D6074 INT  ; 0_1000
B0605_IMP 2603.00 BOOL  ; 10-LITERSIMPULS FRA FLOWMAALER B0605
B0605_LITER D6078 LINT  ; MENGE UT AV T06 I LITER
B0605_MAX_FLOW D6076 INT  ; 0_1000
B201504_PT D6015 CHANNEL  ; NIVAA T20.15    0-1000
B2101_FLT_1 D10100 REAL
B2101_FLT_2 D10102 REAL
B2101_PT D3100 WORD
B2102_FLT_1 D10104 REAL
B2102_FLT_2 D10106 REAL
B2102_PT D3102 WORD
B2103_FLT_1 D10108 REAL
B2103_FLT_2 D10110 REAL
B2103_PT D3104 WORD
B2104_FLT_1 D10112 REAL
B2104_FLT_2 D10114 REAL
B2104_PT D3106 WORD
B2105_NEDSKALERING NEDSKALERING
B2105_TT D3108 WORD
B2106_NEDSKALERING NEDSKALERING
B2106_TT D3110 WORD
B2107_NEDSKALERING NEDSKALERING
B2107_TT D3112 WORD
B2107_TT_HJ D3136 WORD  ; D3112 +/- 0,5 GRADER
B2108_FLOW 4502.15 BOOL
B2108_FLOW_ERVERDI D8112 UINT
B2108_FT D3114 WORD
B2108_FT_L_PR_T D4170 WORD  ; 0-20000
B2108_MENGDE_INN D1672 CHANNEL
B2108_NEDSKALER NEDSKALERING
B2110_HL 2600.14 BOOL  ; Z
B2110_LL 2600.15 BOOL
B2114_PT_FLT2 D10122 REAL
B2115_PT D3164 UINT  ; 0-7,00BAR
B2115_PT_FLT1 D10090 REAL
B2115_PT_FLT2 D10092 REAL
B2119_FL D6160 REAL  ; 0-1000,00
B2119_FLOW D6164 REAL  ; 0-20000 LITERPR TIME
B2119_FL_INN D6158 WORD  ; 0-1000
B2119_NEDSKALERING NEDSKALERING
B2120_FLOW D3590 INT  ; 0-1000
B2120_FLOW_NEDSKALER NEDSKALERING
B2120_FORV_OPNAADD 4802.12 BOOL
B2120_IMP 2603.14 BOOL  ; MAALER PLASSERT VED SJAKT
B2120_MENGDE D3624 DINT  ; MENGDE I LITER
B2120_RESET 4802.11 BOOL  ; RESET MENGDE UT PAA LINJE
B2121_0_7BAR D3156 REAL
B2121_0_7_BAR D3154 REAL
B2121_NEDSKALERING NEDSKALERING
B2121_PT D3160 WORD  ; TRYKK MELLOM P2103 OG SEP21
B2121_PT_FLT D3166 REAL  ; 0-1000
B2121_PT_FLT1 D10116 REAL
B2121_PT_FLT2 D10118 REAL
B2121_PT_mB D3176 INT
B2201_PT D3200 INT
B2201_PT_FLT1 D10030 REAL
B2201_PT_FLT2 D10032 REAL
B2202_PT D3202 INT
B2202_PT_FLT1 D10034 REAL
B2202_PT_FLT2 D10036 REAL
B2203_PT D3204 INT
B2203_PT_FLT1 D10038 REAL
B2203_PT_FLT2 D10040 REAL
B2204_PT D3206 INT
B2204_PT_FLT1 D10042 REAL
B2204_PT_FLT2 D10044 REAL
B2205_NEDSKALERING NEDSKALERING
B2205_TT D3208 WORD
B2205_TT_INVERTERT D23014 WORD  ; TIL BRUK I REG V2252
B2206_NEDSKALERING NEDSKALERING
B2206_TT D3210 WORD
B2207_NEDSKALERING NEDSKALERING
B2207_TT D3212 WORD
B2207_TT_HJ D3256 WORD  ; D3212 +/- 0,5 GRADER
B2208_FT D3214 WORD  ; 0-1000
B2208_FT_L_PR_T D4270 WORD  ; 0-20000
B2208_MENGDE_INN D1674 CHANNEL
B2209_NEDSKALERING NEDSKALERING
B2209_TT D3312 WORD
B2210_HL 2601.14 BOOL  ; Z
B2210_LL 2601.15 BOOL
B2212_PT D3770 DINT
B2212_PT_FLT1 D10046 REAL
B2212_PT_FLT2 D10048 REAL
B2213_PT D3772 DINT
B2213_PT_FLT1 D10050 REAL
B2213_PT_FLT2 D10052 REAL
B2214_PT D3180 INT
B2214_PT_FLT1 D10124 REAL
B2214_PT_FLT2 D10126 REAL
B2215_PT D3298 UINT
B2215_PT_FLT1 D10086 REAL
B2215_PT_FLT2 D10088 REAL
B2219_FL D6260 REAL  ; 0-1000,00
B2219_FLOW D6264 REAL  ; 0-20000 LITERPR TIME
B2219_FL_INN D6258 WORD  ; 0-1000
B2219_NEDSKALERING NEDSKALERING
B2220_FLOW D3592 INT  ; 0-1000
B2220_FLOW_NEDSKALERING NEDSKALERING
B2220_FORV_OPNAADD 4812.12 BOOL
B2220_IMP 2603.15 BOOL  ; MAALER PLASSERT VED SJAKT
B2220_MENGDE D3724 DINT  ; MENGDE I LITER
B2220_RESET 4812.11 BOOL  ; RESET MENGDE UT PAA LINJE
B2302_NEDSKALER NEDSKALERING
B2302_TT D3774 INT
B2305_NEDSKALERING NEDSKALERING
B2305_TT D3300 WORD
B2306_NEDSKALERING NEDSKALERING
B2306_TT D3302 WORD
B2307_NEDSKALERING NEDSKALERING
B2307_TT D3304 WORD
B2307_TT_HJ D3366 WORD  ; D3212 +/- 0,5 GRADER
B2308_FT D3306 WORD
B2308_FT_L_PR_T D4370 WORD  ; 0-8000
B2308_MENGDE_INN D1676 CHANNEL
B2310_NEDSKALER NEDSKALERING
B2310_PT D3308 WORD
B2311_HL_BLK 2603.06 BOOL
B2312_LL_BLK 2603.07 BOOL
B2320_PT D3776 DINT
B2320_PT_FLT1 D10054 REAL
B2320_PT_FLT2 D10056 REAL
B2321_PT D3778 DINT
B2321_PT_FLT1 D10058 REAL
B2321_PT_FLT2 D10060 REAL
B2322_PT D3780 DINT
B2322_PT_FLT1 D10062 REAL
B2322_PT_FLT2 D10064 REAL
B2323_PT D3782 DINT
B2323_PT_FLT1 D10066 REAL
B2323_PT_FLT2 D10068 REAL
B2324_PT D3784 DINT
B2324_PT_FLT1 D10070 REAL
B2324_PT_FLT2 D10072 REAL
B2325_PT D3786 DINT
B2325_PT_FLT1 D10074 REAL
B2325_PT_FLT2 D10076 REAL
B2326_PT D3788 DINT
B2326_PT_FLT1 D10078 REAL
B2326_PT_FLT2 D10080 REAL
B2327_PT D3790 DINT
B2327_PT_FLT1 D10082 REAL
B2327_PT_FLT2 D10084 REAL
B2330_Nedskaler NEDSKALERING
B2330_TT D3792 INT
B2331_BLK_LOKK 2603.05 BOOL
B2332_NEDSKALLERING NEDSKALERING
B2332_TT D3796 INT  ; TEMP VANNKRETS I PAST.REGULERINGSSLOEYFE
B2333_NEDAKALERING NEDSKALERING
B2333_TT D3794 INT
B2360_LL 2603.08 BOOL
B2401_LL 2603.04 BOOL
B2404_NEDSKALERING NEDSKALERING
B2404_PT D3310 WORD
B270102_LL 2603.10 BOOL
B2702_HL 2600.04 BOOL
B2702_LL 2600.05 BOOL
B2703_HL 2600.06 BOOL
B2703_LL 2600.07 BOOL
B4001_LL 2602.13 BOOL
B4002_HL 2602.12 BOOL
B4003_PT_T2740 D1860 CHANNEL  ; 0-1000
B4003_PT_T2740_RAA D1850 CHANNEL
B4004_TT_T2740 D1862 CHANNEL  ; 0-1000
B4004_TT_T2740_RAA D1852 CHANNEL
B4101_LL 2602.15 BOOL
B4102_HL 2602.14 BOOL
B4103_PT_T2741 D1864 CHANNEL  ; 0-1000
B4103_PT_T2741_RAA D1854 CHANNEL
B4104_TT_T2741 D1866 CHANNEL  ; 0-1000
B4104_TT_T2741_RAA D1856 CHANNEL
B4301_SLKONT_PR2 5117.06 BOOL  ; SLANGEKONTROLL TRAKT 42
B8011_CT D1606 REAL  ; Z COND. RET. KURS1 VST80
B8012_TT D1612 REAL  ; Z RETURTEMP VST80 KURS1
B8013_FC 2601.02 BOOL  ; Z
B8014_TT D1600 REAL  ; Z TEMP-TUR. KURS1 VST80
B8015_FC 2601.05 BOOL  ; Z
B8021_CT D1608 REAL  ; Z COND. RET. KURS2 VST80
B8022_TT D1614 REAL  ; Z RETURTEMP VST80 KURS2
B8023_FC 2601.03 BOOL  ; Z
B8024_TT D1602 REAL  ; Z TEMP-TUR. KURS2 VST80
B8025_FC 2601.06 BOOL  ; Z
B8031_CT D1610 REAL  ; Z COND. RET. KURS3 VST80
B8032_TT D1616 REAL  ; Z RETURTEMP VST80 KURS3
B8033_FC 2601.04 BOOL  ; Z
B8034_TT D1604 REAL  ; Z TEMP-TUR. KURS3 VST80
B8035_FC 2601.07 BOOL  ; Z
B8041_CT D1638 REAL  ; Z
B8045_FC 2601.08 BOOL  ; Z
B8101_PT D1634 REAL  ; Z
B8101_TEMP_T81 D1648 REAL
B8201_PT D1628 REAL  ; Z
B8202_TT D1630 REAL  ; Z
B8203_CT D1632 REAL  ; Z
B8301_PT D1622 REAL  ; Z
B8302_TT D1624 REAL  ; Z
B8303_CT D1626 REAL  ; Z
B8401_PT D1618 REAL  ; Z
B8402_TT D1620 REAL  ; Z
B8403_COND D1646 REAL
B8403_CT D1636 REAL  ; Z
B8403_INN 5563 INT
BANE1_GEIT 1451.04 BOOL  ; VED START AV VASK BANE1,VIL VANNVENTIL Vx30 SPERRES OG TIDEN I TR3 SPERRES    x=1-2-3
BANE2_GEIT 1452.04 BOOL  ; VED START AV VASK BANE2,VIL VANNVENTIL Vx30 SPERRES OG TIDEN I TR3 SPERRES      x=1-2-3
BANE3_GEIT 1453.04 BOOL  ; VED START AV VASK BANE3,VIL VANNVENTIL Vx30 SPERRES OG TIDEN I TR3 SPERRES      x=1-2-3
BIL01_0_STATUS 520.01 BOOL  ; XN4_BIL1_. Alle objekter som ikke betjenes er ok
BIL01_1_STATUS 520.02 BOOL  ; XN4_BIL1_. Alle utstyrte objekter i 1.fase er ok
BIL01_2_STAT 520.03 BOOL  ; X Alle utstyrte objekter er ok. Pgm = ok.
BIL01_DRIFT 520.00 BOOL  ; XN4_BIL1_ i drift
BIL01_FEIL 520.04 BOOL  ; XFeil
BIL01_FEILTID 520.05 BOOL  ; X
BIL01_HJ0 420.04 BOOL  ; X
BIL01_HJ1 420.05 BOOL  ; X
BIL01_INDIVID_INNE 520.15 BOOL  ; XIndividadresse er
BIL01_INDKON 520.06 BOOL  ; XKontr. at bare en individadresse er hoey.
BIL01_KOELES 320.14 BOOL  ; SPERR INNLESNING TIL KOE-REGISTER.
BIL01_KOEPLASS_1 D5200 CHANNEL  ; XFOERST I KOE
BIL01_KOEPLASS_2 D5202 CHANNEL  ; X
BIL01_KOEPLASS_3 D5204 CHANNEL  ; X
BIL01_KOMMANDO_KOE 320.15 BOOL  ; D3000 VERDI KAN OVERFOERES TIL KOE-REGISTER.
BIL01_OFF_IMP 520.14 BOOL  ; X
BIL01_ONIMPULS 520.11 BOOL  ; XN4_BIL1_Startimpuls for  program
BIL01_RESET 520.09 BOOL  ; XN4_BIL1. Stopp og nedkobling av programmet
BIL01_START 520.07 BOOL  ; Xprogram starter
BIL01_STARTIMPULS 520.10 BOOL  ; XN4_BIL1. Startimpuls.
BIL01_T03_IND 1220.00 BOOL  ; X
BIL01_T04_IND 1220.01 BOOL  ; XN4_BIL1_TIL_T04_INDIVID
BIL01_T05_IND 1220.02 BOOL  ; X
BIL01_TID_S T0520 BOOL  ; X
BIL01_TID_T 520 NUMBER
BIL01_TIL_T03_VALG 320.00 BOOL  ; INDIVIDVALG FRA KOEREGISTER.
BIL01_TIL_T04_VALG 320.01 BOOL  ; INDIVIDVALG FRA KOEREGISTER.
BIL01_TIL_T05_VALG 320.02 BOOL  ; INDIVIDVALG FRA KOEREGISTER.
BIL01_TMU_USIKRET 520.08 BOOL  ; TMU
BIL02_0_STATUS 522.01 BOOL  ; XN4_BIL1_. Alle objekter som ikke betjenes er ok
BIL02_1_STATUS 522.02 BOOL  ; XN4_BIL1_. Alle utstyrte objekter i 1.fase er ok
BIL02_2_STAT 522.03 BOOL  ; X Alle utstyrte objekter er ok. Pgm = ok.
BIL02_DRIFT 522.00 BOOL  ; XN4_BIL1_ i drift
BIL02_FEIL 522.04 BOOL  ; XFeil
BIL02_FEILTID 522.05 BOOL  ; X
BIL02_HJ0 422.04 BOOL  ; X
BIL02_HJ1 422.05 BOOL  ; X
BIL02_INDIVID_INNE 522.15 BOOL  ; XIndividadresse er
BIL02_INDKON 522.06 BOOL  ; XKontr. at bare en individadresse er hoey.
BIL02_KOEINLES D5228 CHANNEL  ; XINNLESNING AVKOMMANDOVERDIER FRA D3000
BIL02_KOELES 322.14 BOOL  ; SPERR INNLESNING TIL KOE-REGISTER.
BIL02_KOEPLASS_1 D5220 CHANNEL  ; XFOERST I KOE
BIL02_KOEPLASS_2 D5222 CHANNEL  ; X
BIL02_KOEPLASS_3 D5224 CHANNEL  ; X
BIL02_KOEPLASS_4 D5226 CHANNEL  ; X
BIL02_KOMMANDO_KOE 322.15 BOOL  ; D3000 VERDI KAN OVERFOERES TIL KOE-REGISTER.
BIL02_OFF_IMP 522.14 BOOL  ; X
BIL02_ONIMPULS 522.11 BOOL  ; XN4_BIL1_Startimpuls for  program
BIL02_RESET 522.09 BOOL  ; XN4_BIL1. Stopp og nedkobling av programmet
BIL02_START 522.07 BOOL  ; Xprogram starter
BIL02_STARTIMPULS 522.10 BOOL  ; XN4_BIL1. Startimpuls.
BIL02_T03_IND 1222.00 BOOL  ; X
BIL02_T04_IND 1222.01 BOOL  ; XN4_BIL1_TIL_T04_INDIVID
BIL02_T05_IND 1222.02 BOOL  ; X
BIL02_TID_S T0522 BOOL  ; X
BIL02_TID_T 522 NUMBER
BIL02_TIL_T03_VALG 322.00 BOOL  ; INDIVIDVALG FRA KOEREGISTER.
BIL02_TIL_T04_VALG 322.01 BOOL  ; INDIVIDVALG FRA KOEREGISTER.
BIL02_TIL_T05_VALG 322.02 BOOL  ; XINDIVIDVALG FRA KOEREGISTER.
BK_21_NIVAA D3158 CHANNEL
BK_22_NIVAA D3248 CHANNEL
BLAASETID_FOR T0009 BOOL
BLIK_TID1_S T0871 BOOL
BLIK_TID2_S T0872 BOOL
BLINK 999.01 BOOL  ; 0,5 SEKUNERS BINK
BLINK_HURTIG T0895 BOOL  ; 0.2S BLINK
BRYTER_HJ 960.15 BOOL
BUS_BLAAS_LAB 2824.02 BOOL
BUS_BLAAS_UHT 2824.03 BOOL
BUS_KNAPP_V4302 2935.05 BOOL
BUS_SIGN_VACUUM 2824.01 BOOL
Betinget_Omslag_DP3 202.01 BOOL
C01_IND_VST80_K1 1200.00 BOOL  ; Z
C01_STATUS D7620 CHANNEL  ; VASKESTATUS
C01_TYPE_VASK D7600 CHANNEL  ; VALG AV VASK SE EGEN TABELL
C01_VALG_VST80_K1 300.00 BOOL  ; Z
C02_IND_VST80_K1 1200.03 BOOL  ; Z
C02_STATUS D7623 CHANNEL  ; VASKESTATUS
C02_TYPE_VASK D7603 CHANNEL  ; VALG AV VASK SE EGEN TABELL
C02_VALG_VST80_K1 300.03 BOOL  ; Z
C03_06_C81_SYRE 1454.11 BOOL  ; VASKES BARE MED SYRE
C03_07_C81_FORL_FASE 1454.00 BOOL
C03_07_C81_HETVANN 1454.12 BOOL
C03_07_C81_LUT_SYRE 1454.10 BOOL
C03_07_C81_NOEDSTOPP 1454.02 BOOL
C03_07_C81_STOPP_TUR 1454.01 BOOL
C03_IND_VST80_K2 1201.00 BOOL  ; Z
C03_STATUS D7720 CHANNEL  ; VASKESTATUS
C03_TYPE_VASK D7700 CHANNEL  ; VALG AV VASK SE EGEN TABELL
C03_VALG_VST80_K2 301.00 BOOL  ; Z
C05_IND_VST80_K2 1201.03 BOOL  ; Z
C05_STATUS D7723 CHANNEL  ; VASKESTATUS
C05_TYPE_VASK D7703 CHANNEL  ; VALG AV VASK SE EGEN TABELL
C05_VALG_VST80_K2 301.03 BOOL  ; Z
C06_IND_VST80_K2 1201.06 BOOL  ; Z
C06_STATUS D7726 CHANNEL  ; VASKESTATUS
C06_TYPE_VASK D7706 CHANNEL  ; VALG AV VASK SE EGEN TABELL
C06_VALG_VST80_K2 301.06 BOOL  ; Z
C07_IND_VST80_K2 1201.07 BOOL  ; Z
C07_STATUS D7727 CHANNEL  ; VASKESTATUS
C07_TYPE_VASK D7707 CHANNEL  ; VALG AV VASK SE EGEN TABELL
C07_VALG_VST80_K2 301.07 BOOL
C08_IND_VST80_K2 1201.08 BOOL  ; Z
C08_STATUS D7728 CHANNEL  ; VASKESTATUS
C08_TYPE_VASK D7708 CHANNEL  ; VALG AV VASK SE EGEN TABELL
C08_VALG_VST80_K2 301.08 BOOL  ; Z
C09_0_ST_HJ1 933.07 BOOL
C09_0_ST_HJ2 933.08 BOOL
C09_0_ST_HJ3 933.09 BOOL
C09_0_ST_HJ4 933.10 BOOL
C09_10_0_ST_HJ1 933.15 BOOL
C09_10_15_2_HJ1 936.03 BOOL
C09_1_HJ1 935.01 BOOL
C09_1_HJ2 935.02 BOOL
C09_C10_1_HJ1 935.05 BOOL
C09_IND_VST80_K3 1202.04 BOOL  ; Z
C09_STATUS D7824 CHANNEL  ; VASKESTATUS
C09_TYPE_VASK D7804 CHANNEL  ; VALG AV VASK SE EGEN TABELL
C09_VALG 302.04 BOOL
C10_0_ST_HJ1 933.11 BOOL
C10_0_ST_HJ2 933.12 BOOL
C10_0_ST_HJ3 933.13 BOOL
C10_0_ST_HJ4 933.14 BOOL
C10_1_HJ1 935.03 BOOL
C10_1_HJ2 935.04 BOOL
C10_IND_VST80_K3 1202.05 BOOL  ; Z
C10_STATUS D7825 CHANNEL  ; VASKESTATUS
C10_TYPE_VASK D7805 CHANNEL  ; VALG AV VASK SE EGEN TABELL
C10_VALG 302.05 BOOL
C12_1_HJ1 935.06 BOOL
C12_1_HJ2 935.07 BOOL
C12_C33_36_1_HJ1 935.09 BOOL
C12_IND_VST80_K3 1202.00 BOOL  ; Z
C12_STATUS D7820 CHANNEL  ; VASKESTATUS
C12_TYPE_VASK D7800 CHANNEL  ; VALG AV VASK SE EGEN TABELL
C12_VALG 302.00 BOOL  ; Z
C13_1_HJ1 935.10 BOOL
C13_1_HJ2 935.11 BOOL
C13_34_37_1_HJ1 935.13 BOOL
C13_IND_VST80_K3 1202.01 BOOL  ; Z
C13_STATUS D7821 CHANNEL  ; VASKESTATUS
C13_TYPE_VASK D7801 CHANNEL  ; VALG AV VASK SE EGEN TABELL
C13_VALG 302.01 BOOL  ; Z
C14_1_HJ1 935.14 BOOL
C14_1_HJ2 935.15 BOOL
C14_C35_38_1_HJ1 936.01 BOOL
C14_IND_VST80_K3 1202.02 BOOL  ; Z
C14_STATUS D7822 CHANNEL  ; VASKESTATUS
C14_TYPE_VASK D7802 CHANNEL  ; VALG AV VASK SE EGEN TABELL
C14_VALG 302.02 BOOL  ; Z
C15_1_HJ1 936.04 BOOL
C15_1_HJ2 936.05 BOOL
C15_1_HJ3 940.01 BOOL
C15_HJ1 934.04 BOOL
C15_HJ2 934.09 BOOL
C15_HJ3 934.10 BOOL
C15_HJ4 934.15 BOOL
C15_IND_VST80_K3 1202.06 BOOL  ; Z
C15_STATUS D7826 CHANNEL  ; VASKESTATUS
C15_TYPE_VASK D7806 CHANNEL  ; VALG AV VASK SE EGEN TABELL
C15_VALG 302.06 BOOL  ; Z
C17_DRE_ETTER_C_N6 2842.01 BOOL
C18_DRE_ETTER_C_N6 2842.02 BOOL
C19_DRE_ETTER_C_N6 2842.03 BOOL
C20_DRE_ETTER_C_N6 2842.04 BOOL
C21_DREN_STARTET 760.00 BOOL
C21_DREN_UTFOERT 760.01 BOOL
C21_LITER_PRS_UT D3640 UDINT
C21_STARTET 760.02 BOOL
C21_UTFOERT 760.03 BOOL
C22_LITER_PRS_UT D3740 UDINT
C23_ACC_FORSK_TID D3321 WORD
C23_ACC_HETV_SIRK_TID D3341 WORD
C23_ACC_LUTSIRK_TID D3325 WORD
C23_ACC_LUTSKYLL_TID D3329 WORD
C23_ACC_SYRESIRK_TID D3333 WORD
C23_ACC_SYRESKYLL_TID D3337 WORD
C23_AV_BLK_FYLL 4504.14 BOOL  ; SIGNAL SOM SKAL BENYTTES  VED OPPFYLING AV BLK ETTER VASK.
C23_AV_BLK_FYLL_S T0887 BOOL  ; SIGNAL SOM SKAL BENYTTES  VED OPPFYLING AV BLK ETTER VASK.
C23_AV_BLK_FYLL_T 0887 NUMBER
C23_FORLENG_FASE 4504.07 BOOL  ; PAST21
C23_FORSKYLL 4503.01 BOOL  ; PAST21
C23_FORSKYLLTELLER_C C0086 BOOL
C23_FORSKYLLTELLER_S C86 CHANNEL
C23_FORST_TIL_VST80 4504.12 BOOL  ; PAST21  PAST22 OG 23 MAA VENTE
C23_HJ_LUTSKYLL_LUT_TID D3330 WORD
C23_HJ_REG_FORSK_TID D3322 WORD
C23_HJ_REG_HETV_SIRK_TID D3342 WORD
C23_HJ_REG_LUTSIRK_TID D3326 WORD
C23_HJ_REG_SYRESIRK_TID D3334 WORD
C23_HJ_REG_SYRESKYLL_TID D3338 WORD
C23_KLAP_ER_TRINNTELLER D3640 INT
C23_KLAP_ER_TRINNTELLER_N5 2845 INT
C23_KLAP_ER_TRINNTID D3636 INT
C23_KLAP_INNE_VST80_K4 4504.15 BOOL
C23_KLAP_PRS_TRINNTELLER D3638 INT
C23_KLAP_PRS_TRINNTID D3634 INT
C23_LUTSIRK_TID_S T0094 BOOL
C23_LUTSIRK_TID_T 0094 NUMBER
C23_LUT_INN 4503.09 BOOL  ; PAST21
C23_LUT_INN_KONS_1 4503.10 BOOL  ; PAST21
C23_LUT_SIRK 4503.11 BOOL  ; PAST21
C23_LUT_SKYLL 4503.14 BOOL  ; PAST21
C23_LUT_SYRE 4504.10 BOOL  ; PAST21
C23_LUT_UT 4503.12 BOOL  ; PAST21
C23_LUT_UT_KONS_0 4503.13 BOOL  ; PAST21
C23_PROD_TEKST D3622 INT  ; TIL GRAFIKK
C23_PRS_FORSK_MENGDE D3344 WORD
C23_PRS_FORSK_TID D3320 WORD  ; D3321
C23_PRS_HETV_SIRK_TID D3340 WORD
C23_PRS_LUTSIRK_TID D3324 WORD
C23_PRS_LUTSKYLL_TID D3328 WORD
C23_PRS_SYRESIRK_TID D3332 WORD
C23_PRS_SYRESKYLL_TID D3336 WORD
C23_RAP_COND_LUT D9158 CHANNEL  ; VASKERAPPORT CONDUKTIVITET I LUTFASEN
C23_RAP_COND_SYRE D9164 CHANNEL  ; VASKERAPPORT COND. I SYRESIRK. I SEKUNDER
C23_RAP_FLOW D9190 CHANNEL  ; VASKERAPPORT  FLOW I L/T
C23_RAP_HJ_COND_LUT D9159 CHANNEL  ; VASKERAPPORT CONDUKTIVITET I LUTFASEN HJ.FUNK.
C23_RAP_HJ_COND_SYRE D9165 CHANNEL  ; VASKERAPPORT CONDUKTIVITET I SYREFASEN HJ.FUNK.
C23_RAP_HJ_TEMP_HETV D9171 CHANNEL  ; VASKERAPPORT TEMP.HETVANNSIRK. HJ_FUNKSJON
C23_RAP_HJ_TEMP_LUT D9157 CHANNEL  ; VASKERAPPORT TEMP UT AV PASTEUR  I LUTFASEN HJ_FUNKSJON
C23_RAP_HJ_TEMP_SYRE D9163 CHANNEL  ; VASKERAPPORT TEMP UT AV PASTEUR ISYREFASEN HJ_FUNKSJON
C23_RAP_SEK_FS D9150 CHANNEL  ; VASKERAPPORT TID I FORSKYLLING I SEKUNDER
C23_RAP_SEK_LUT D9154 CHANNEL  ; VASKERAPPORT TID I LUTSIRK. I SEKUNDER
C23_RAP_SEK_SYRE D9160 CHANNEL  ; VASKERAPPORT TID I FORSKYLLING I SEKUNDER
C23_RAP_STATUS D9166 CHANNEL  ; ¨
C23_RAP_TEMP_HETV D9170 CHANNEL  ; VASKERAPPORT TEMP.HETVANNSIRK.
C23_RAP_TEMP_LUT D9156 CHANNEL  ; VASKERAPPORT TEMP UT AV PASTEUR  I LUTFASEN
C23_RAP_TEMP_SYRE D9162 CHANNEL  ; VASKERAPPORT TEMP UT AV PASTEUR ISYREFASEN
C23_RAP_TID_HETV D9168 CHANNEL  ; VASKERAPPORT TID HETVANNSIRK.
C23_STERILISER 4504.11 BOOL  ; PAST21
C23_STERIL_AVSLUTT 4504.01 BOOL  ; PAST21
C23_STERIL_OPPVARM 4503.15 BOOL
C23_STERIL_SIRK 4504.00 BOOL  ; PAST21
C23_STERIL_V2104_LAV_TEMP 4504.04 BOOL  ; PAST21
C23_STOPP_ETTER_VM 4504.09 BOOL  ; PAST21
C23_STOPP_I_FASE 4504.08 BOOL  ; PAST21 STANSER PUMPER OG TILFOERSEL BAV LUT-SYRE
C23_SYRE_INN 4503.03 BOOL  ; PAST21
C23_SYRE_INN_KONS_1 4503.04 BOOL  ; PAST21
C23_SYRE_MED_FORSKYLL 4504.06 BOOL  ; PAST21
C23_SYRE_SIRK 4503.05 BOOL  ; PAST21
C23_SYRE_SKYLL 4503.08 BOOL  ; PAST21
C23_SYRE_UT 4503.06 BOOL  ; PAST21
C23_SYRE_UT_KONS_0 4503.07 BOOL  ; PAST21
C23_TEKST_BILDE D4042 CHANNEL
C23_V2104_LAV_TEMP 4504.05 BOOL  ; PAST21
C23_VASKEPGM_DRIFT 4503.00 BOOL  ; PAST21 FORLOEP INNE
C23_VASKERAPP_OK 4505.03 BOOL
C23_VASKETRINN_TEKST D3620 INT
C23_VASK_ENDE 4504.13 BOOL  ; SIGNAL SOM SKAL BENYTTES  VED OPPFYLING AV BLK ETTER VASK
C23_VENT_INN_UT_VASKEM 4503.02 BOOL  ; 450303
C24_ACC_FORSK_TID D3421 WORD
C24_ACC_HETV_SIRK_TID D3441 WORD
C24_ACC_LUTSIRK_TID D3425 WORD
C24_ACC_LUTSKYLL_TID D3429 WORD
C24_ACC_SYRESIRK_TID D3433 WORD
C24_ACC_SYRESKYLL_TID D3437 WORD
C24_AV_BLK_FYLL 4514.14 BOOL  ; SIGNAL SOM SKAL BENYTTES  VED OPPFYLING AV BLK ETTER VASK.
C24_AV_BLK_FYLL_S T0888 BOOL  ; SIGNAL SOM SKAL BENYTTES  VED OPPFYLING AV BLK ETTER VASK.
C24_AV_BLK_FYLL_T 0888 NUMBER
C24_ER_FORSK_MENGDE D3446 WORD
C24_FORLENG_FASE 4514.07 BOOL  ; PAST22
C24_FORSKYLL 4513.01 BOOL  ; PAST22
C24_FORST_TIL_VST80 4514.12 BOOL  ; PAST22  PAST21 OG 23 MAA VENTE
C24_HC_HOY_FLOW 4814.04 BOOL
C24_HC_HOY_FLOW_AV 4814.05 BOOL  ; ¨
C24_HC_HOY_FLOW_REG_VERDI D3750 INT  ; AKTUELL RESTTID I AKTUELL FASE
C24_HJ_LUTSKYLL_LUT_TID D3430 WORD
C24_HJ_REG_FORSK_TID D3422 WORD
C24_HJ_REG_HETV_SIRK_TID D3442 WORD
C24_HJ_REG_LUTSIRK_TID D3426 WORD
C24_HJ_REG_SYRESIRK_TID D3434 WORD
C24_HJ_REG_SYRESKYLL_TID D3438 WORD
C24_KLAP_ER_TRINNTELLER D3760 INT
C24_KLAP_ER_TRINNTID D3756 INT
C24_KLAP_INNE_VST80_K4 4514.15 BOOL
C24_KLAP_PRS_TRINNTELLER D3758 INT
C24_KLAP_PRS_TRINNTID D3754 INT
C24_LUT_INN 4513.09 BOOL  ; ¨
C24_LUT_INN_KONS_1 4513.10 BOOL  ; PAST22
C24_LUT_SIRK 4513.11 BOOL  ; PAST22
C24_LUT_SKYLL 4513.14 BOOL  ; PAST22
C24_LUT_SYRE 4514.10 BOOL  ; PAST22
C24_LUT_UT 4513.12 BOOL  ; PAST22
C24_LUT_UT_KONS_0 4513.13 BOOL  ; PAST22
C24_PROD_TEKST D3722 INT  ; TIL  GRAFIKK
C24_PRS_FORSK_MENGDE D3444 WORD
C24_PRS_FORSK_TID D3420 WORD
C24_PRS_HETV_SIRK_TID D3440 WORD
C24_PRS_LUTSIRK_TID D3424 WORD
C24_PRS_LUTSKYLL_TID D3428 WORD
C24_PRS_SYRESIRK_TID D3432 WORD
C24_PRS_SYRESKYLL_TID D3436 WORD
C24_RAP_COND_LUT D9258 CHANNEL  ; VASKERAPPORT CONDUKTIVITET I LUTFASEN
C24_RAP_COND_SYRE D9264 CHANNEL  ; VASKERAPPORT COND. I SYRESIRK. I SEKUNDER
C24_RAP_FLOW D9290 CHANNEL  ; VASKERAPPORT  FLOW I L/T
C24_RAP_HJ_COND_LUT D9259 CHANNEL  ; VASKERAPPORT CONDUKTIVITET I LUTFASEN HJ.FUNK.
C24_RAP_HJ_COND_SYRE D9265 CHANNEL  ; VASKERAPPORT CONDUKTIVITET I SYREFASEN HJ.FUNK.
C24_RAP_HJ_TEMP_HETV D9271 CHANNEL  ; VASKERAPPORT TEMP.HETVANNSIRK. HJ_FUNKSJON
C24_RAP_HJ_TEMP_LUT D9257 CHANNEL  ; VASKERAPPORT TEMP UT AV PASTEUR  I LUTFASEN HJ_FUNKSJON
C24_RAP_HJ_TEMP_SYRE D9263 CHANNEL  ; VASKERAPPORT TEMP UT AV PASTEUR ISYREFASEN HJ_FUNKSJON
C24_RAP_SEK_FS D9250 CHANNEL  ; VASKERAPPORT TID I FORSKYLLING I SEKUNDER
C24_RAP_SEK_LUT D9254 CHANNEL  ; VASKERAPPORT TID I LUTSIRK. I SEKUNDER
C24_RAP_SEK_SYRE D9260 CHANNEL  ; VASKERAPPORT TID I FORSKYLLING I SEKUNDER
C24_RAP_STATUS D9266 CHANNEL  ; VASKERAPPORT STATUS          0=GODKJ.  1=DRIFTFORS.  2= IKKE GODKJ.
C24_RAP_TEMP_HETV D9270 CHANNEL  ; VASKERAPPORT TEMP.HETVANNSIRK.
C24_RAP_TEMP_LUT D9256 CHANNEL  ; VASKERAPPORT TEMP UT AV PASTEUR  I LUTFASEN
C24_RAP_TEMP_SYRE D9262 CHANNEL  ; VASKERAPPORT TEMP UT AV PASTEUR ISYREFASEN
C24_RAP_TID_HETV D9268 CHANNEL  ; VASKERAPPORT TID HETVANNSIRK.
C24_STERILISER 4514.11 BOOL  ; PAST22
C24_STERIL_AVSLUTT 4514.01 BOOL  ; PAST22
C24_STERIL_OPPVARM 4513.15 BOOL  ; PAST22
C24_STERIL_SIRK 4514.00 BOOL  ; PAST22
C24_STOPP_ETTER_VM 4514.09 BOOL  ; PAST22
C24_STOPP_I_FASE 4514.08 BOOL  ; PAST22   STANSER PUMPER OG TILFOERSEL BAV LUT-SYRE
C24_SYRE_INN 4513.03 BOOL  ; PAST22
C24_SYRE_INN_KONS_1 4513.04 BOOL  ; PAST22
C24_SYRE_MED_FORSKYLL 4514.06 BOOL  ; ¨
C24_SYRE_SIRK 4513.05 BOOL  ; PAST22
C24_SYRE_SKYLL 4513.08 BOOL  ; PAST22
C24_SYRE_UT 4513.06 BOOL  ; PAST22
C24_SYRE_UT_KONS_0 4513.07 BOOL  ; PAST22
C24_TEKST_BILDE D4192 CHANNEL
C24_TMU_HC_HOY_FLOW 4814.06 BOOL
C24_VASKEPGM_DRIFT 4513.00 BOOL  ; PAST22  FORLOEP INNE
C24_VASKERAPP_OK 4515.03 BOOL
C24_VASKETRINN_TEKST D3720 INT
C24_VASK_ENDE 4514.13 BOOL  ; SIGNAL SOM SKAL BENYTTES  VED OPPFYLING AV BLK ETTER VASK
C24_VENT_INN_UT_VASKEM 4513.02 BOOL  ; PAST22   PAST2 ELLER PAST23 FYLLES-TOEMMES FOR VASKEMIDDEL
C254_KLAP_INNE_VST80_K4 4514.15 BOOL
C25_ACC_FORSK_TID D3521 WORD
C25_ACC_HETV_SIRK_TID D3541 WORD
C25_ACC_LUTSIRK_TID D3525 WORD
C25_ACC_LUTSKYLL_TID D3529 WORD
C25_ACC_SYRESIRK_TID D3533 WORD
C25_ACC_SYRESKYLL_TID D3537 WORD
C25_AVSLUTTET 4824.01 BOOL
C25_AV_BLK_FYLL 4524.14 BOOL  ; SIGNAL SOM SKAL BENYTTES  VED OPPFYLING AV BLK ETTER VASK.
C25_AV_BLK_FYLL_S T0889 BOOL  ; SIGNAL SOM SKAL BENYTTES  VED OPPFYLING AV BLK ETTER VASK.
C25_AV_BLK_FYLL_T 0889 NUMBER
C25_BLK_NIV 4824.00 BOOL  ; V2309 STENGES
C25_ER_FORSK_MENGDE D3546 WORD
C25_FORLENG_FASE 4524.07 BOOL  ; PAST23
C25_FORSKYLL 4523.01 BOOL  ; PAST23
C25_FORST_TIL_VST80 4524.12 BOOL  ; PAST23  PAST21 OG 22 MAA VENTE
C25_HJ_LUTSKYLL_LUT_TID D3530 WORD
C25_HJ_REG_FORSK_TID D3522 WORD
C25_HJ_REG_HETV_SIRK_TID D3542 WORD
C25_HJ_REG_LUTSIRK_TID D3526 WORD
C25_HJ_REG_SYRESIRK_TID D3534 WORD
C25_HJ_REG_SYRESKYLL_TID D3538 WORD
C25_IND_VST80_K4 1205.00 BOOL  ; VASK PAST23
C25_KLAP_ER_TRINNTELLER D3860 INT
C25_KLAP_ER_TRINNTID D3856 INT
C25_KLAP_INNE_VST80_K4 4524.15 BOOL
C25_KLAP_PRS_TRINNTELLER D3858 INT
C25_KLAP_PRS_TRINNTID D3854 INT
C25_LUT_INN 4523.09 BOOL  ; PAST23
C25_LUT_INN_KONS_1 4523.10 BOOL  ; PAST23
C25_LUT_SIRK 4523.11 BOOL  ; PAST23
C25_LUT_SKYLL 4523.14 BOOL  ; PAST23
C25_LUT_SYRE 4524.10 BOOL  ; PAST23
C25_LUT_UT 4523.12 BOOL  ; PAST23
C25_LUT_UT_KONS_0 4523.13 BOOL  ; ¨
C25_PROD_TEKST D3822 INT  ; TIL  GRAFIKK
C25_PRS_FORSK_MENGDE D3544 WORD
C25_PRS_FORSK_TID D3520 WORD
C25_PRS_HETV_SIRK_TID D3540 WORD
C25_PRS_LUTSIRK_TID D3524 WORD  ; ¨
C25_PRS_LUTSKYLL_TID D3528 WORD
C25_PRS_SYRESIRK_TID D3532 WORD
C25_PRS_SYRESKYLL_TID D3536 WORD
C25_RAP_COND_LUT D9358 CHANNEL  ; VASKERAPPORT CONDUKTIVITET I LUTFASEN
C25_RAP_COND_SYRE D9364 CHANNEL  ; VASKERAPPORT COND. I SYRESIRK. I SEKUNDER
C25_RAP_FLOW D9390 CHANNEL  ; VASKERAPPORT  FLOW I L/T
C25_RAP_HJ_COND_LUT D9359 CHANNEL  ; VASKERAPPORT CONDUKTIVITET I LUTFASEN HJ.FUNK.
C25_RAP_HJ_COND_SYRE D9365 CHANNEL  ; VASKERAPPORT CONDUKTIVITET I SYREFASEN HJ.FUNK.
C25_RAP_HJ_TEMP_HETV D9371 CHANNEL  ; VASKERAPPORT TEMP.HETVANNSIRK. HJ_FUNKSJON
C25_RAP_HJ_TEMP_LUT D9357 CHANNEL  ; VASKERAPPORT TEMP UT AV PASTEUR  I LUTFASEN HJ_FUNKSJON
C25_RAP_HJ_TEMP_SYRE D9363 CHANNEL  ; VASKERAPPORT TEMP UT AV PASTEUR ISYREFASEN HJ_FUNKSJON
C25_RAP_SEK_FS D9350 CHANNEL  ; VASKERAPPORT TID I FORSKYLLING I SEKUNDER
C25_RAP_SEK_LUT D9354 CHANNEL  ; VASKERAPPORT TID I LUTSIRK. I SEKUNDER
C25_RAP_SEK_SYRE D9360 CHANNEL  ; VASKERAPPORT TID I FORSKYLLING I SEKUNDER
C25_RAP_STATUS D9366 CHANNEL  ; VASKERAPPORT STATUS          0=GODKJ.  1=DRIFTFORS.  2= IKKE GODKJ.
C25_RAP_TEMP_HETV D9370 CHANNEL  ; VASKERAPPORT TEMP.HETVANNSIRK.
C25_RAP_TEMP_LUT D9356 CHANNEL  ; VASKERAPPORT TEMP UT AV PASTEUR  I LUTFASEN
C25_RAP_TEMP_SYRE D9362 CHANNEL  ; VASKERAPPORT TEMP UT AV PASTEUR ISYREFASEN
C25_RAP_TID_HETV D9368 CHANNEL  ; VASKERAPPORT TID HETVANNSIRK.
C25_STERILISER 4524.11 BOOL  ; PAST23
C25_STERIL_AVSLUTT 4524.01 BOOL  ; PAST23
C25_STERIL_OPPVARM 4523.15 BOOL  ; PAST23
C25_STERIL_SIRK 4524.00 BOOL  ; PAST23
C25_STOPP_ETTER_VM 4524.09 BOOL  ; PAST23
C25_STOPP_I_FASE 4524.08 BOOL  ; PAST23   STANSER PUMPER OG TILFOERSEL BAV LUT-SYRE
C25_SYRE_INN 4523.03 BOOL  ; ¨
C25_SYRE_INN_KONS_1 4523.04 BOOL  ; PAST23
C25_SYRE_MED_FORSKYLL 4524.06 BOOL  ; PAST23
C25_SYRE_SIRK 4523.05 BOOL  ; PAST23
C25_SYRE_SKYLL 4523.08 BOOL  ; PAST23
C25_SYRE_UT 4523.06 BOOL  ; PAST23
C25_SYRE_UT_KONS_0 4523.07 BOOL  ; PAST23
C25_TEKST_BILDE D4292 CHANNEL
C25_TEMP_OK 4524.05 BOOL  ; PAST23
C25_VASKEPGM_DRIFT 4523.00 BOOL  ; ¨
C25_VASKERAPP_OK 4525.03 BOOL
C25_VASKETRINN_TEKST D3820 INT
C25_VASK_ENDE 4524.13 BOOL  ; SIGNAL SOM SKAL BENYTTES  VED OPPFYLING AV BLK ETTER VASK
C25_VENT_INN_UT_VASKEM 4523.02 BOOL  ; PAST23   PAST2 ELLER PAST22FYLLES-TOEMMES FOR VASKEMIDDEL
C30_IND_VST80_K3 1202.03 BOOL  ; Z
C30_STATUS D7823 CHANNEL  ; VASKESTATUS
C30_TYPE_VASK D7803 CHANNEL  ; VALG AV VASK SE EGEN TABELL
C30_VALG 302.03 BOOL  ; Z
C31_IND_VST80_K1 1200.05 BOOL  ; Z
C31_STATUS D7625 CHANNEL  ; VASKESTATUS
C31_TYPE_VASK D7605 CHANNEL  ; VALG AV VASK SE EGEN TABELL
C31_VALG_VST80_K1 300.05 BOOL  ; Z
C32_IND_VST80_K2 1201.05 BOOL  ; Z
C32_STATUS D7725 CHANNEL  ; VASKESTATUS
C32_TYPE_VASK D7705 CHANNEL  ; VALG AV VASK SE EGEN TABELL
C32_VALG_VST80_K2 301.05 BOOL  ; Z
C33_36_1_HJ1 935.08 BOOL
C33_IND_VST80_K3 1202.07 BOOL  ; ¨
C33_STATUS D7827 CHANNEL  ; VASKESTATUS
C33_TYPE_VASK D7807 CHANNEL  ; VALG AV VASK SE EGEN TABELL
C33_VALG 302.07 BOOL  ; Z
C34_37_1_HJ1 935.12 BOOL
C34_IND_VST80_K3 1202.08 BOOL  ; Z
C34_STATUS D7828 CHANNEL  ; VASKESTATUS
C34_TYPE_VASK D7808 CHANNEL  ; VALG AV VASK SE EGEN TABELL
C34_VALG 302.08 BOOL  ; Z
C35_38_1_HJ1 936.00 BOOL
C35_IND_VST80_K3 1202.09 BOOL  ; Z
C35_STATUS D7829 CHANNEL  ; VASKESTATUS
C35_TYPE_VASK D7809 CHANNEL  ; VALG AV VASK SE EGEN TABELL
C35_VALG 302.09 BOOL
C36_IND_VST80_K3 1202.10 BOOL  ; Z
C36_STATUS D7830 CHANNEL  ; VASKESTATUS
C36_TYPE_VASK D7810 CHANNEL  ; VALG AV VASK SE EGEN TABELL
C36_VALG 302.10 BOOL  ; Z
C37_IND_VST80_K3 1202.11 BOOL  ; Z
C37_STATUS D7831 CHANNEL  ; VASKESTATUS
C37_TYPE_VASK D7811 CHANNEL  ; VALG AV VASK SE EGEN TABELL
C37_VALG 302.11 BOOL  ; Z
C38_IND_VST80_K3 1202.12 BOOL
C38_STATUS D7832 CHANNEL  ; VASKESTATUS
C38_TYPE_VASK D7812 CHANNEL  ; VALG AV VASK SE EGEN TABELL
C38_VALG 302.12 BOOL  ; Z
C50_IND_VST80_K2 1201.09 BOOL  ; Z
C50_STATUS D7729 CHANNEL  ; VASKESTATUS
C50_TYPE_VASK D7709 CHANNEL  ; VALG AV VASK SE EGEN TABELL
C50_VALG_VST80_K2 301.09 BOOL  ; Z
C52_IND_VST80_K2 1201.10 BOOL  ; Z
C52_STATUS D7730 CHANNEL  ; VASKESTATUS
C52_TYPE_VASK D7710 CHANNEL  ; VALG AV VASK SE EGEN TABELL
C52_VALG_VST80_K2 301.10 BOOL  ; Z
C53_IND_VST80_K2 1201.11 BOOL  ; Z
C53_STATUS D7731 CHANNEL  ; VASKESTATUS
C53_TYPE_VASK D7711 CHANNEL  ; VALG AV VASK SE EGEN TABELL
C53_VALG_VST80_K2 301.11 BOOL  ; Z
C54_IND_VST80_K2 1201.12 BOOL  ; Z
C54_STATUS D7732 CHANNEL  ; VASKESTATUS
C54_TYPE_VASK D7712 CHANNEL  ; VALG AV VASK SE EGEN TABELL
C54_VALG_VST80_K2 301.12 BOOL  ; Z
C77_IND_VST80_K2 1201.13 BOOL  ; Z
C77_STATUS D7733 CHANNEL  ; VASKESTATUS
C77_TYPE_VASK D7713 CHANNEL  ; VALG AV VASK SE EGEN TABELL
C77_VALG_VST80_K2 301.13 BOOL  ; Z
C78_IND_VST80_K2 1201.14 BOOL  ; Z
C78_STATUS D7734 CHANNEL  ; VASKESTATUS
C78_TYPE_VASK D7714 CHANNEL  ; VALG AV VASK SE EGEN TABELL
C78_VALG_VST80_K2 301.14 BOOL  ; Z
C79_IND_VST80_K2 1201.15 BOOL  ; Z
C79_LAMPE_MOTTTAK 2604.00 BOOL
C79_STATUS D7735 CHANNEL  ; VASKESTATUS
C79_TYPE_VASK D7715 CHANNEL  ; VALG AV VASK SE EGEN TABELL
C79_VALG_VST80_K2 301.15 BOOL
C80_FEIL_TIL_PLS1_GR2860 4612.05 BOOL  ; INVERTERT
C80_FORL_FASE 1450.00 BOOL  ; 150100
C80_HETVANN 1450.12 BOOL
C80_K2_KLAPRETRINN_N5 2840 INT  ; KLAPRETRINN FRA VST80 K2
C80_KLAPRETRINN 4634 INT  ; KLAPRETRINN FRA VST80 K1-K2-K3
C80_LUT_SYRE 1450.10 BOOL
C80_NOEDSTOPP 1450.02 BOOL
C80_STOPP_TUR 1450.01 BOOL
C80_SYRE 1450.11 BOOL  ; VASKES BARE MED SYRE
C81_IND_VST80_K1 1200.01 BOOL  ; Z
C81_SOM_CONAINERVASK 2603.13 BOOL
C81_STATUS D7621 CHANNEL  ; VASKESTATUS
C81_TYPE_VASK D7601 CHANNEL  ; VALG AV VASK SE EGEN TABELL
C81_VALG_VST80_K1 300.01 BOOL  ; Z
C82_IND_VST80_K1 1200.04 BOOL  ; Z
C82_STATUS D7624 CHANNEL  ; VASKESTATUS
C82_TYPE_VASK D7604 CHANNEL  ; VALG AV VASK SE EGEN TABELL
C82_VALGT_VST80_K1 300.04 BOOL  ; Z
C83_IND_VST80_K2 1201.01 BOOL  ; Z
C83_STATUS D7721 CHANNEL  ; VASKESTATUS
C83_TYPE_VASK D7701 CHANNEL  ; VALG AV VASK SE EGEN TABELL
C83_VALG_VST80_K2 301.01 BOOL  ; Z
C84_IND_VST80_K2 1201.04 BOOL  ; Z
C84_STATUS D7724 CHANNEL  ; VASKESTATUS
C84_TYPE_VASK D7704 CHANNEL  ; VALG AV VASK SE EGEN TABELL
C84_VALG_VST80_K2 301.04 BOOL  ; Z
C85_IND_VST80_K1 1200.02 BOOL  ; Z
C85_STATUS D7622 CHANNEL  ; VASKESTATUS
C85_TYPE_VASK D7602 CHANNEL  ; VALG AV VASK SE EGEN TABELL
C85_VALG_VST80_K1 300.02 BOOL  ; Z
C86_IND_VST80_K2 1201.02 BOOL  ; Z
C86_STATUS D7722 CHANNEL  ; VASKESTATUS
C86_TYPE_VASK D7702 CHANNEL  ; VALG AV VASK SE EGEN TABELL
C86_VALG_VST80_K2 301.02 BOOL  ; Z
C95_FORL_FASE 1455.00 BOOL
C95_HETVANN 1455.12 BOOL
C95_LUT_SYRE 1455.10 BOOL
C95_NOEDSTOPP 1455.02 BOOL
C95_STOPP_TUR 1455.01 BOOL
C95_SYRE 1455.11 BOOL  ; VASKES BARE MED SYRE
C_B1_H1_VEKSL_TR1_S T0401 BOOL  ; V8047 OG 8048 VEKSLES I C81-84
C_B1_H1_VEKSL_TR1_T 0401 NUMBER  ; V8047 OG 8048 VEKSLES I C81-84
C_B1_H1_VEKSL_TR2_S T0402 BOOL  ; V8047 OG 8048 VEKSLES I C81-84
C_B1_H1_VEKSL_TR2_T 0402 NUMBER  ; V8047 OG 8048 VEKSLES I C81-84
C_B1_H1_VEKSL_TR3_S T0403 BOOL  ; V8047 OG 8048 VEKSLES I C81-84
C_B1_H1_VEKSL_TR3_T 0403 NUMBER  ; V8047 OG 8048 VEKSLES I C81-84
C_B1_H1_VEKSL_TR4_S T0404 BOOL  ; V8047 OG 8048 VEKSLES I C81-84
C_B1_H1_VEKSL_TR4_T 0404 NUMBER  ; V8047 OG 8048 VEKSLES I C81-84
C_B2_H2_VEKSL_TR1_S T0405 BOOL  ; V8053 OG 8054 VEKSLES I C82 OG C83
C_B2_H2_VEKSL_TR1_T 0405 NUMBER  ; V8053 OG 8054 VEKSLES I C82 OG C83
C_B2_H2_VEKSL_TR2_S T0406 BOOL  ; V8053 OG 8054 VEKSLES I C82 OG C83
C_B2_H2_VEKSL_TR2_T 0406 NUMBER  ; V8053 OG 8054 VEKSLES I C82 OG C83
C_B2_H2_VEKSL_TR3_S T0407 BOOL  ; V8053 OG 8054 VEKSLES I C82 OG C83
C_B2_H2_VEKSL_TR3_T 0407 NUMBER  ; V8053 OG 8054 VEKSLES I C82 OG C83
C_B2_H2_VEKSL_TR4_S T0408 BOOL  ; V8053 OG 8054 VEKSLES I C82 OG C83
C_B2_H2_VEKSL_TR4_T 0408 NUMBER  ; V8053 OG 8054 VEKSLES I C82 OG C83
C_BANE1_FEIL 501.04 BOOL
C_BANE1_FEIL_TIL_PLS1_GR2870 4612.13 BOOL  ; INVERTERT
C_BANE1_FORL_FASE 1451.00 BOOL
C_BANE1_HETVANN 1451.12 BOOL
C_BANE1_LUT_SYRE 1451.10 BOOL
C_BANE1_NOEDSTOPP 1451.02 BOOL
C_BANE1_STOPP_TUR 1451.01 BOOL
C_BANE1_SYRE 1451.11 BOOL  ; VASKES BARE MED SYRE
C_BANE2_FEIL 502.04 BOOL
C_BANE2_FEIL_TIL_PLS1_GR2880 4613.05 BOOL  ; INVERTERT
C_BANE2_FORL_FASE 1452.00 BOOL  ; 145400
C_BANE2_HETVANN 1452.12 BOOL
C_BANE2_LUT_SYRE 1452.10 BOOL
C_BANE2_NOEDSTOPP 1452.02 BOOL
C_BANE2_STOPP_TUR 1452.01 BOOL
C_BANE2_SYRE 1452.11 BOOL  ; VASKES BARE MED SYRE
C_BANE3_FEIL_TIL_PLS1_GR2890 4613.13 BOOL  ; INVERTERT
C_BANE3_FORL_FASE 1453.00 BOOL
C_BANE3_HETVANN 1453.12 BOOL
C_BANE3_LUT_SYRE 1453.10 BOOL
C_BANE3_NOEDSTOPP 1453.02 BOOL
C_BANE3_STOPP_TUR 1453.01 BOOL
C_BANE3_SYRE 1453.11 BOOL  ; VASKES BARE MED SYRE
C_KURS3_2_STATUS 502.03 BOOL
C_SILO_2_HJ1 936.02 BOOL
C_SILO_FEIL_TIL_PLS1_GR3000 4614.05 BOOL  ; INVERTERT
C_SILO_VEKSL_RV_TV 502.13 BOOL  ; C36-37-38  NAAR 502.13=1 ER VASKEN MAKEN TIL C33-34-35.   NAAR 502.13=0 ER VASKEN MAKEN  TIL C12-13-14
C_T03_05_HJ1 935.00 BOOL
C_T03_HJ1 934.00 BOOL
C_T03_HJ2 934.01 BOOL
C_T03_HJ3 934.02 BOOL
C_T03_HJ4 934.03 BOOL
C_T04_HJ1 934.05 BOOL
C_T04_HJ2 934.06 BOOL
C_T04_HJ3 934.07 BOOL
C_T04_HJ4 934.08 BOOL
C_T05_HJ1 934.11 BOOL
C_T05_HJ2 934.12 BOOL
C_T05_HJ3 934.13 BOOL
C_T05_HJ4 934.14 BOOL
C_T05_HJ5 934.15 BOOL
Copy_of_P21_DP2_OK_UTFORS_T 0804 NUMBER
Copy_of_PAST21_FLOETE_V_T2401_T 0829 NUMBER  ; FLOETE VED T24.01
Copy_of_PAST23_FLOTE_INN_T 0840 NUMBER  ; FORSINK SINAL FLOETE I BLK
Copy_of_SCAN_INN_KONTR_T 0842 NUMBER  ; 1_SCAN_FORSINKER
D3800_RESET 4825.15 BOOL  ; NOE UKLART
DIVISOR_INNGANGSORD D3020 REAL  ; DELER INGANGSVERDI MED 32,760 FOR OMREGNING TIL 0-1000
DREN_P2028_N5 2916.01 BOOL
DREN_P2029_N5 2916.02 BOOL
DREN_P2031_N5 2916.03 BOOL
DREN_P2044_N5 2916.04 BOOL
DREN_UHT_START_PUMPER 2915.00 BOOL
DRIFT1_DOS_T82 1402.06 BOOL  ; Drift dosering vaskemiddel. T 82 Luttank.
DRIFT1_DOS_T83 1403.06 BOOL  ; Drift dosering vaskemiddel. T 83 Syretank.
DRIFT1_DOS_T84 1404.06 BOOL
DRIFT_DOS_T82 1402.05 BOOL  ; Drift dosering vaskemiddel. T 82 Luttank.
DRIFT_DOS_T83 1403.05 BOOL  ; Drift dosering vaskemiddel. T 83 Syretank.
DRIFT_DOS_T84 1404.05 BOOL
DUMMY 1999.00 BOOL
Dummy 3041.00 BOOL
FEILRESET 999.00 BOOL  ; XRESET AV FEIL I NODE 4.
FEILRESET_TIL_N5 2800.00 BOOL
FEILTID_VACUUM T0911 BOOL
FEIL_VACUUM 2806.01 BOOL
FORSINK_KOND_K1_S T0111 BOOL
FORSINK_KOND_K2_S T0121 BOOL
FORSINK_TEMPFEIL_K1 T0036 BOOL
FORSINK_TEMPFEIL_K2 T0136 BOOL
FORSINK_TEMPFEIL_K3 T0236 BOOL
FORSINK_V4302 T0004 BOOL
FORS_CONDFEIL_K1 T0035 BOOL
FORS_CONDFEIL_K2 T0135 BOOL
FORS_CONDFEIL_K3 T0235 BOOL
FORS_SPJELDTID T0008 BOOL
FORS_VDREN_L11 720.04 BOOL
FORS_VDREN_L12 720.12 BOOL
FORS_VDREN_L21 722.04 BOOL
FORS_VDREN_L22 722.12 BOOL
FOR_SLUK_TANK 2904.11 BOOL
GR27_LA_LAB_V_PR2 5010.00 BOOL  ; LAMPE UHT. VED TRAKT FOR GRISEFOR.       C79ER INNKOBLET
GR27_LA_UHT_V_PR2 5010.01 BOOL  ; LAMPE LAB VED TRAKT FOR GRISEFOR.       C79 ER INNKOBLET
GR520_1_HJ1 936.12 BOOL
GR521_1_HJ1 937.03 BOOL
GR522_1_HJ1 937.10 BOOL
GR523_1_HJ1 938.01 BOOL
GR524_1_HJ0 424.04 BOOL  ; X
GR524_1_HJ1 938.08 BOOL
GR524_2_HJ0 424.05 BOOL  ; ER 1 NAAR DET ER KLART TIL PASTEURENE
GR525_1_HJ0 425.04 BOOL  ; X
GR525_1_HJ1 938.15 BOOL
GR525_2_HJ0 425.05 BOOL  ; ER 1 NAAR DET ER KLART TIL PASTEURENE
H4_1_2_01_AUTO 1600.00 BOOL  ; HOVEDTAVLE 4.1_SEKSJON_SKUFF        DRIFTSIGN. FRA  NODE1_4
H4_1_2_01_AUTO_PR2 5000.00 BOOL  ; HOVEDTAVLE 4.1_SEKSJON_SKUFF        DRIFTSIGN. FRA  NODE1_4
H4_1_2_01_FEIL 1600.01 BOOL  ; HOVEDTAVLE 4.1_SEKSJON_SKUFF        UTLOEST MOTORV. ELLER SIKRING
H4_1_2_01_FEIL_PR2 5100.01 BOOL  ; HOVEDTAVLE 4.1_SEKSJON_SKUFF        UTLOEST MOTORV. ELLER SIKRING
H4_1_2_01_OK 1600.02 BOOL  ; HOVEDTAVLE 4.1_SEKSJON_SKUFF       DRIFT OG OK
H4_1_2_01_OK_PR2 5100.00 BOOL  ; HOVEDTAVLE 4.1_SEKSJON_SKUFF       DRIFT OG OK
H4_1_2_02_AUTO 1600.03 BOOL  ; HOVEDTAVLE 4.1_SEKSJON_SKUFF        DRIFTSIGN. FRA  NODE1_4
H4_1_2_02_AUTO_PR2 5000.01 BOOL  ; HOVEDTAVLE 4.1_SEKSJON_SKUFF        DRIFTSIGN. FRA  NODE1_4
H4_1_2_02_FEIL 1600.04 BOOL  ; HOVEDTAVLE 4.1_SEKSJON_SKUFF        UTLOEST MOTORV. ELLER SIKRING
H4_1_2_02_FEIL_PR2 5100.03 BOOL  ; HOVEDTAVLE 4.1_SEKSJON_SKUFF        UTLOEST MOTORV. ELLER SIKRING
H4_1_2_02_OK 1600.05 BOOL  ; HOVEDTAVLE 4.1_SEKSJON_SKUFF       DRIFT OG OK
H4_1_2_02_OK_PR2 5100.02 BOOL  ; HOVEDTAVLE 4.1_SEKSJON_SKUFF       DRIFT OG OK
H4_1_2_03_AUTO 1600.06 BOOL  ; HOVEDTAVLE 4.1_SEKSJON_SKUFF        DRIFTSIGN. FRA  NODE1_4
H4_1_2_03_AUTO_PR2 5000.02 BOOL  ; HOVEDTAVLE 4.1_SEKSJON_SKUFF        DRIFTSIGN. FRA  NODE1_4
H4_1_2_03_FEIL 1600.07 BOOL  ; HOVEDTAVLE 4.1_SEKSJON_SKUFF        UTLOEST MOTORV. ELLER SIKRING
H4_1_2_03_FEIL_PR2 5100.05 BOOL  ; HOVEDTAVLE 4.1_SEKSJON_SKUFF        UTLOEST MOTORV. ELLER SIKRING
H4_1_2_03_OK 1600.08 BOOL  ; HOVEDTAVLE 4.1_SEKSJON_SKUFF       DRIFT OG OK
H4_1_2_03_OK_PR2 5100.04 BOOL  ; HOVEDTAVLE 4.1_SEKSJON_SKUFF       DRIFT OG OK
H4_1_2_04_AUTO 1600.09 BOOL  ; HOVEDTAVLE 4.1_SEKSJON_SKUFF        DRIFTSIGN. FRA  NODE1_4
H4_1_2_04_AUTO_PR2 5000.03 BOOL  ; HOVEDTAVLE 4.1_SEKSJON_SKUFF        DRIFTSIGN. FRA  NODE1_4
H4_1_2_04_FEIL 1600.10 BOOL  ; HOVEDTAVLE 4.1_SEKSJON_SKUFF        UTLOEST MOTORV. ELLER SIKRING
H4_1_2_04_FEIL_PR2 5100.07 BOOL  ; HOVEDTAVLE 4.1_SEKSJON_SKUFF        UTLOEST MOTORV. ELLER SIKRING
H4_1_2_04_OK 1600.11 BOOL  ; HOVEDTAVLE 4.1_SEKSJON_SKUFF       DRIFT OG OK
H4_1_2_04_OK_PR2 5100.06 BOOL  ; HOVEDTAVLE 4.1_SEKSJON_SKUFF       DRIFT OG OK
H4_1_2_05_AUTO 1600.12 BOOL  ; HOVEDTAVLE 4.1_SEKSJON_SKUFF        DRIFTSIGN. FRA  NODE1_4
H4_1_2_05_AUTO_PR2 5000.04 BOOL  ; HOVEDTAVLE 4.1_SEKSJON_SKUFF        DRIFTSIGN. FRA  NODE1_4
H4_1_2_05_FEIL 1600.13 BOOL  ; HOVEDTAVLE 4.1_SEKSJON_SKUFF        UTLOEST MOTORV. ELLER SIKRING
H4_1_2_05_FEIL_PR2 5101.01 BOOL  ; HOVEDTAVLE 4.1_SEKSJON_SKUFF        UTLOEST MOTORV. ELLER SIKRING
H4_1_2_05_OK 1600.14 BOOL  ; HOVEDTAVLE 4.1_SEKSJON_SKUFF       DRIFT OG OK
H4_1_2_05_OK_PR2 5101.00 BOOL  ; HOVEDTAVLE 4.1_SEKSJON_SKUFF       DRIFT OG OK
H4_1_2_06_AUTO 1601.00 BOOL  ; HOVEDTAVLE 4.1_SEKSJON_SKUFF        DRIFTSIGN. FRA  NODE1_4
H4_1_2_06_AUTO_PR2 5000.05 BOOL  ; HOVEDTAVLE 4.1_SEKSJON_SKUFF        DRIFTSIGN. FRA  NODE1_4
H4_1_2_06_FEIL 1601.01 BOOL  ; HOVEDTAVLE 4.1_SEKSJON_SKUFF        UTLOEST MOTORV. ELLER SIKRING
H4_1_2_06_FEIL_PR2 5101.03 BOOL  ; HOVEDTAVLE 4.1_SEKSJON_SKUFF        UTLOEST MOTORV. ELLER SIKRING
H4_1_2_06_OK 1601.02 BOOL  ; HOVEDTAVLE 4.1_SEKSJON_SKUFF       DRIFT OG OK
H4_1_2_06_OK_PR2 5101.02 BOOL  ; HOVEDTAVLE 4.1_SEKSJON_SKUFF       DRIFT OG OK
H4_1_2_07_AUTO 1601.03 BOOL  ; HOVEDTAVLE 4.1_SEKSJON_SKUFF        DRIFTSIGN. FRA  NODE1_4
H4_1_2_07_AUTO_PR2 5000.06 BOOL  ; HOVEDTAVLE 4.1_SEKSJON_SKUFF        DRIFTSIGN. FRA  NODE1_4
H4_1_2_07_FEIL 1601.04 BOOL  ; HOVEDTAVLE 4.1_SEKSJON_SKUFF        UTLOEST MOTORV. ELLER SIKRING
H4_1_2_07_FEIL_PR2 5101.05 BOOL  ; HOVEDTAVLE 4.1_SEKSJON_SKUFF        UTLOEST MOTORV. ELLER SIKRING
H4_1_2_07_OK 1601.05 BOOL  ; HOVEDTAVLE 4.1_SEKSJON_SKUFF       DRIFT OG OK
H4_1_2_07_OK_PR2 5101.04 BOOL  ; HOVEDTAVLE 4.1_SEKSJON_SKUFF       DRIFT OG OK
H4_1_2_08_AUTO 1601.06 BOOL  ; HOVEDTAVLE 4.1_SEKSJON_SKUFF        DRIFTSIGN. FRA  NODE1_4
H4_1_2_08_AUTO_PR2 5000.07 BOOL  ; HOVEDTAVLE 4.1_SEKSJON_SKUFF        DRIFTSIGN. FRA  NODE1_4
H4_1_2_08_FEIL 1601.07 BOOL  ; HOVEDTAVLE 4.1_SEKSJON_SKUFF        UTLOEST MOTORV. ELLER SIKRING
H4_1_2_08_FEIL_PR2 5101.07 BOOL  ; HOVEDTAVLE 4.1_SEKSJON_SKUFF        UTLOEST MOTORV. ELLER SIKRING
H4_1_2_08_OK 1601.08 BOOL  ; HOVEDTAVLE 4.1_SEKSJON_SKUFF       DRIFT OG OK
H4_1_2_08_OK_PR2 5101.06 BOOL  ; HOVEDTAVLE 4.1_SEKSJON_SKUFF       DRIFT OG OK
H4_1_2_09_AUTO 1601.09 BOOL  ; HOVEDTAVLE 4.1_SEKSJON_SKUFF        DRIFTSIGN. FRA  NODE1_4
H4_1_2_09_AUTO_PR2 5001.00 BOOL  ; HOVEDTAVLE 4.1_SEKSJON_SKUFF        DRIFTSIGN. FRA  NODE1_4
H4_1_2_09_FEIL 1601.10 BOOL  ; HOVEDTAVLE 4.1_SEKSJON_SKUFF        UTLOEST MOTORV. ELLER SIKRING
H4_1_2_09_FEIL_PR2 5102.01 BOOL  ; HOVEDTAVLE 4.1_SEKSJON_SKUFF        UTLOEST MOTORV. ELLER SIKRING
H4_1_2_09_OK 1601.11 BOOL  ; HOVEDTAVLE 4.1_SEKSJON_SKUFF       DRIFT OG OK
H4_1_2_09_OK_PR2 5102.00 BOOL  ; HOVEDTAVLE 4.1_SEKSJON_SKUFF       DRIFT OG OK
H4_1_2_10_AUTO 1601.12 BOOL  ; HOVEDTAVLE 4.1_SEKSJON_SKUFF        DRIFTSIGN. FRA  NODE1_4
H4_1_2_10_AUTO_PR2 5001.01 BOOL  ; HOVEDTAVLE 4.1_SEKSJON_SKUFF        DRIFTSIGN. FRA  NODE1_4
H4_1_2_10_FEIL 1601.13 BOOL  ; HOVEDTAVLE 4.1_SEKSJON_SKUFF        UTLOEST MOTORV. ELLER SIKRING
H4_1_2_10_FEIL_PR2 5102.03 BOOL  ; HOVEDTAVLE 4.1_SEKSJON_SKUFF        UTLOEST MOTORV. ELLER SIKRING
H4_1_2_10_OK 1601.14 BOOL  ; HOVEDTAVLE 4.1_SEKSJON_SKUFF       DRIFT OG OK
H4_1_2_10_OK_PR2 5102.02 BOOL  ; HOVEDTAVLE 4.1_SEKSJON_SKUFF       DRIFT OG OK
H4_1_3_01_AUTO 1602.00 BOOL  ; HOVEDTAVLE 4.1_SEKSJON_SKUFF        DRIFTSIGN. FRA  NODE1_4
H4_1_3_01_AUTO_PR2 5002.00 BOOL  ; HOVEDTAVLE 4.1_SEKSJON_SKUFF        DRIFTSIGN. FRA  NODE1_4
H4_1_3_01_FEIL 1602.01 BOOL  ; HOVEDTAVLE 4.1_SEKSJON_SKUFF        UTLOEST MOTORV. ELLER SIKRING
H4_1_3_01_FEIL_PR2 5103.01 BOOL  ; HOVEDTAVLE 4.1_SEKSJON_SKUFF        UTLOEST MOTORV. ELLER SIKRING
H4_1_3_01_OK 1602.02 BOOL  ; HOVEDTAVLE 4.1_SEKSJON_SKUFF       DRIFT OG OK
H4_1_3_01_OK_PR2 5103.00 BOOL  ; HOVEDTAVLE 4.1_SEKSJON_SKUFF       DRIFT OG OK
H4_1_3_02_AUTO 1602.03 BOOL  ; HOVEDTAVLE 4.1_SEKSJON_SKUFF        DRIFTSIGN. FRA  NODE1_4
H4_1_3_02_AUTO_PR2 5002.01 BOOL  ; HOVEDTAVLE 4.1_SEKSJON_SKUFF        DRIFTSIGN. FRA  NODE1_4
H4_1_3_02_FEIL 1602.04 BOOL  ; HOVEDTAVLE 4.1_SEKSJON_SKUFF        UTLOEST MOTORV. ELLER SIKRING
H4_1_3_02_FEIL_PR2 5103.03 BOOL  ; HOVEDTAVLE 4.1_SEKSJON_SKUFF        UTLOEST MOTORV. ELLER SIKRING
H4_1_3_02_OK 1602.05 BOOL  ; HOVEDTAVLE 4.1_SEKSJON_SKUFF       DRIFT OG OK
H4_1_3_02_OK_PR2 5103.02 BOOL  ; HOVEDTAVLE 4.1_SEKSJON_SKUFF       DRIFT OG OK
H4_1_3_03_AUTO 1602.06 BOOL  ; HOVEDTAVLE 4.1_SEKSJON_SKUFF        DRIFTSIGN. FRA  NODE1_4
H4_1_3_03_AUTO_PR2 5002.02 BOOL  ; HOVEDTAVLE 4.1_SEKSJON_SKUFF        DRIFTSIGN. FRA  NODE1_4
H4_1_3_03_FEIL 1602.07 BOOL  ; HOVEDTAVLE 4.1_SEKSJON_SKUFF        UTLOEST MOTORV. ELLER SIKRING
H4_1_3_03_FEIL_PR2 5103.05 BOOL  ; HOVEDTAVLE 4.1_SEKSJON_SKUFF        UTLOEST MOTORV. ELLER SIKRING
H4_1_3_03_OK 1602.08 BOOL  ; HOVEDTAVLE 4.1_SEKSJON_SKUFF       DRIFT OG OK
H4_1_3_03_OK_PR2 5103.04 BOOL  ; HOVEDTAVLE 4.1_SEKSJON_SKUFF       DRIFT OG OK
H4_1_3_04_AUTO 1602.09 BOOL  ; HOVEDTAVLE 4.1_SEKSJON_SKUFF        DRIFTSIGN. FRA  NODE1_4
H4_1_3_04_AUTO_PR2 5002.03 BOOL  ; HOVEDTAVLE 4.1_SEKSJON_SKUFF        DRIFTSIGN. FRA  NODE1_4
H4_1_3_04_FEIL 1602.10 BOOL  ; HOVEDTAVLE 4.1_SEKSJON_SKUFF        UTLOEST MOTORV. ELLER SIKRING
H4_1_3_04_FEIL_PR2 5103.07 BOOL  ; HOVEDTAVLE 4.1_SEKSJON_SKUFF        UTLOEST MOTORV. ELLER SIKRING
H4_1_3_04_OK 1602.11 BOOL  ; HOVEDTAVLE 4.1_SEKSJON_SKUFF       DRIFT OG OK
H4_1_3_04_OK_PR2 5103.06 BOOL  ; HOVEDTAVLE 4.1_SEKSJON_SKUFF       DRIFT OG OK
H4_1_3_05_AUTO 1602.12 BOOL  ; HOVEDTAVLE 4.1_SEKSJON_SKUFF        DRIFTSIGN. FRA  NODE1_4
H4_1_3_05_AUTO_PR2 5002.04 BOOL  ; HOVEDTAVLE 4.1_SEKSJON_SKUFF        DRIFTSIGN. FRA  NODE1_4
H4_1_3_05_FEIL 1602.13 BOOL  ; HOVEDTAVLE 4.1_SEKSJON_SKUFF        UTLOEST MOTORV. ELLER SIKRING
H4_1_3_05_FEIL_PR2 5104.01 BOOL  ; HOVEDTAVLE 4.1_SEKSJON_SKUFF        UTLOEST MOTORV. ELLER SIKRING
H4_1_3_05_OK 1602.14 BOOL  ; HOVEDTAVLE 4.1_SEKSJON_SKUFF       DRIFT OG OK
H4_1_3_05_OK_PR2 5104.00 BOOL  ; HOVEDTAVLE 4.1_SEKSJON_SKUFF       DRIFT OG OK
H4_1_3_06_AUTO 1603.00 BOOL  ; HOVEDTAVLE 4.1_SEKSJON_SKUFF        DRIFTSIGN. FRA  NODE1_4
H4_1_3_06_AUTO_PR2 5002.05 BOOL  ; HOVEDTAVLE 4.1_SEKSJON_SKUFF        DRIFTSIGN. FRA  NODE1_4
H4_1_3_06_FEIL 1603.01 BOOL  ; HOVEDTAVLE 4.1_SEKSJON_SKUFF        UTLOEST MOTORV. ELLER SIKRING
H4_1_3_06_FEIL_PR2 5104.03 BOOL  ; HOVEDTAVLE 4.1_SEKSJON_SKUFF        UTLOEST MOTORV. ELLER SIKRING
H4_1_3_06_OK 1603.02 BOOL  ; HOVEDTAVLE 4.1_SEKSJON_SKUFF       DRIFT OG OK
H4_1_3_06_OK_PR2 5104.02 BOOL  ; HOVEDTAVLE 4.1_SEKSJON_SKUFF       DRIFT OG OK
H4_1_3_09_AUTO 1603.09 BOOL  ; HOVEDTAVLE 4.1_SEKSJON_SKUFF        DRIFTSIGN. FRA  NODE1_4
H4_1_3_09_AUTO_PR2 5002.06 BOOL  ; HOVEDTAVLE 4.1_SEKSJON_SKUFF        DRIFTSIGN. FRA  NODE1_4
H4_1_3_09_FEIL 1603.10 BOOL  ; HOVEDTAVLE 4.1_SEKSJON_SKUFF        UTLOEST MOTORV. ELLER SIKRING
H4_1_3_09_FEIL_PR2 5104.05 BOOL  ; HOVEDTAVLE 4.1_SEKSJON_SKUFF        UTLOEST MOTORV. ELLER SIKRING
H4_1_3_09_OK 1603.11 BOOL  ; HOVEDTAVLE 4.1_SEKSJON_SKUFF       DRIFT OG OK
H4_1_3_09_OK_PR2 5104.04 BOOL  ; HOVEDTAVLE 4.1_SEKSJON_SKUFF       DRIFT OG OK
H4_1_4_01_AUTO 1604.00 BOOL  ; HOVEDTAVLE 4.1_SEKSJON_SKUFF        DRIFTSIGN. FRA  NODE1_4
H4_1_4_01_AUTO_PR2 5003.00 BOOL  ; HOVEDTAVLE 4.1_SEKSJON_SKUFF        DRIFTSIGN. FRA  NODE1_4
H4_1_4_01_FEIL 1604.01 BOOL  ; HOVEDTAVLE 4.1_SEKSJON_SKUFF        UTLOEST MOTORV. ELLER SIKRING
H4_1_4_01_FEIL_PR2 5105.01 BOOL  ; HOVEDTAVLE 4.1_SEKSJON_SKUFF        UTLOEST MOTORV. ELLER SIKRING
H4_1_4_01_OK 1604.02 BOOL  ; HOVEDTAVLE 4.1_SEKSJON_SKUFF       DRIFT OG OK
H4_1_4_01_OK_PR2 5105.00 BOOL  ; HOVEDTAVLE 4.1_SEKSJON_SKUFF       DRIFT OG OK
H4_1_4_02_AUTO 1604.03 BOOL  ; HOVEDTAVLE 4.1_SEKSJON_SKUFF        DRIFTSIGN. FRA  NODE1_4
H4_1_4_02_AUTO_PR2 5003.01 BOOL  ; HOVEDTAVLE 4.1_SEKSJON_SKUFF        DRIFTSIGN. FRA  NODE1_4
H4_1_4_02_FEIL 1604.04 BOOL  ; HOVEDTAVLE 4.1_SEKSJON_SKUFF        UTLOEST MOTORV. ELLER SIKRING
H4_1_4_02_FEIL_PR2 5105.03 BOOL  ; HOVEDTAVLE 4.1_SEKSJON_SKUFF        UTLOEST MOTORV. ELLER SIKRING
H4_1_4_02_OK 1604.05 BOOL  ; HOVEDTAVLE 4.1_SEKSJON_SKUFF       DRIFT OG OK
H4_1_4_02_OK_PR2 5105.02 BOOL  ; HOVEDTAVLE 4.1_SEKSJON_SKUFF       DRIFT OG OK
H4_1_4_03_AUTO 1604.06 BOOL  ; HOVEDTAVLE 4.1_SEKSJON_SKUFF        DRIFTSIGN. FRA  NODE1_4
H4_1_4_03_AUTO_PR2 5003.02 BOOL  ; HOVEDTAVLE 4.1_SEKSJON_SKUFF        DRIFTSIGN. FRA  NODE1_4
H4_1_4_03_FEIL 1604.07 BOOL  ; HOVEDTAVLE 4.1_SEKSJON_SKUFF        UTLOEST MOTORV. ELLER SIKRING
